(* CoDeSys 2.3 project: esx_ioxp_PPS_gazel.pro *)
(* Libraries: esx_ioxp.lib 19.12.13 13:14:40, Util.lib 18.5.10 15:14:28, Standard.lib 4.10.05 11:14:46 *)

(* PLC configuration (modules and I/O channels)
gq_Ignition AT %IX0.0 [X_SYS_IGNITION] Ignition pin (D+)
gs16_TempBoard AT %IW1 [X_SYS_TEMP_BOARD] System temperature in degree Celsius
gu32_TimeMs AT %ID1 [X_SYS_TIME_MS] System time in ms
gq_StayAlive AT %QX0.0 [X_SYS_STAY_ALIVE] Stay alive mechanism
gq_Relay AT %QX1.0 [X_SYS_RELAY_1] Safety relay
gs32_SensorSupply AT %QD1 [X_SYS_SENSOR_SUPPLY_1] External sensor supply
gs32_IO01 AT %QD2 [InOut] IO01, PIN 9 (PWM H/L, DO, CC, VIN (40V), DIN) {InOut_Type = uninitialized; InOut_FilterConfig = 0; InOut_Circuit1 = X_OUT_CIRCUIT_HIGH_SIDE; InOut_Circuit2 = X_IN_CIRCUIT_NO_PULL_UP; PWM_MaxValue = 10000}
gs32_IO02 AT %QD3 [InOut] ---- GAS meter ---- IO02, PIN 8 (PWM H/L, DO, CC, VIN (40V), DIN) {InOut_Type = X_IN_TYPE_VOLTAGE_40V; InOut_FilterConfig = 0; InOut_Circuit1 = X_IN_CIRCUIT_ACTIVE_HIGH; InOut_Circuit2 = X_IN_CIRCUIT_PULL_UP; PWM_MaxValue = 10000}
gs32_IO03 AT %QD4 [InOut] --- GAS LED BAR  ---  IO03, PIN 7 (PWM H/L, DO, CC, VIN ( {InOut_Type = X_OUT_TYPE_PWM; InOut_FilterConfig = 0; InOut_Circuit1 = X_OUT_CIRCUIT_PUSH_PULL; InOut_Circuit2 = X_IN_CIRCUIT_NO_PULL_UP; PWM_MaxValue = 10000}
gs32_IO04 AT %QD5 [InOut] IO04, PIN 6 (PWM H/L, DO, CC, VIN (40V), DIN) {InOut_Type = X_OUT_TYPE_PWM; InOut_FilterConfig = 0; InOut_Circuit1 = X_OUT_CIRCUIT_HIGH_SIDE; InOut_Circuit2 = X_IN_CIRCUIT_NO_PULL_UP; PWM_MaxValue = 10000}
gs32_IO05 AT %QD6 [InOut] IO05, PIN 13 (PWM H, DO, DIN) {InOut_Type = uninitialized; InOut_FilterConfig = 0; InOut_Circuit1 = X_OUT_CIRCUIT_HIGH_SIDE; InOut_Circuit2 = X_IN_CIRCUIT_NO_PULL_UP; PWM_MaxValue = 10000}
gs32_IO06 AT %QD7 [InOut] ---Inj1--- IO06, PIN 12 (PWM H, DO, DIN) {InOut_Type = X_OUT_TYPE_DIGITAL; InOut_FilterConfig = 0; InOut_Circuit1 = X_OUT_CIRCUIT_HIGH_SIDE; InOut_Circuit2 = X_IN_CIRCUIT_NO_PULL_UP; PWM_MaxValue = 10000}
gs32_IO07 AT %QD8 [InOut] --- Inj2 -----IO07, PIN 11 (PWM H, DO, DIN) {InOut_Type = uninitialized; InOut_FilterConfig = 0; InOut_Circuit1 = X_IN_CIRCUIT_ACTIVE_HIGH; InOut_Circuit2 = X_IN_CIRCUIT_NO_PULL_UP; PWM_MaxValue = 10000}
gs32_IO08 AT %QD9 [InOut] --- PPS1 emul --  IO08, PIN 10 (PWM H, DO, DIN) {InOut_Type = X_OUT_TYPE_PWM; InOut_FilterConfig = 0; InOut_Circuit1 = X_OUT_CIRCUIT_HIGH_SIDE; InOut_Circuit2 = X_IN_CIRCUIT_NO_PULL_UP; PWM_MaxValue = 10000}
gs32_IO09 AT %ID2 [InOut] IO09, PIN 2 (DIN, FIN, IIN) {InOut_Type = uninitialized; InOut_FilterConfig = 0; InOut_Circuit1 = X_IN_CIRCUIT_ACTIVE_HIGH; InOut_Circuit2 = X_IN_CIRCUIT_NO_PULL_UP; PWM_MaxValue = 10000}
gs32_IO10 AT %ID3 [InOut] ---RPM--- IO10, PIN 3 (DIN, FIN, IIN) {InOut_Type = X_IN_TYPE_FREQUENCY; InOut_FilterConfig = 0; InOut_Circuit1 = X_IN_CIRCUIT_ACTIVE_HIGH; InOut_Circuit2 = X_IN_CIRCUIT_NO_PULL_UP; PWM_MaxValue = 10000}
gs32_IO11 AT %ID4 [InOut] IO11, PIN 4 (DIN, FIN, IIN) {InOut_Type = uninitialized; InOut_FilterConfig = 0; InOut_Circuit1 = X_IN_CIRCUIT_ACTIVE_HIGH; InOut_Circuit2 = X_IN_CIRCUIT_NO_PULL_UP; PWM_MaxValue = 10000}
gs32_IO12 AT %ID5 [InOut] ---BLOCK ON--- IO12, PIN 5 (DIN) {InOut_Type = X_IN_TYPE_DIGITAL; InOut_FilterConfig = 0; InOut_Circuit1 = X_IN_CIRCUIT_ACTIVE_HIGH; InOut_Circuit2 = X_IN_CIRCUIT_NO_PULL_UP; PWM_MaxValue = 10000}
gs32_IO13 AT %ID6 [InOut] IO13, PIN 38 (CIN (20mA), DIN) {InOut_Type = uninitialized; InOut_FilterConfig = 0; InOut_Circuit1 = X_IN_CIRCUIT_ACTIVE_HIGH; InOut_Circuit2 = X_IN_CIRCUIT_NO_PULL_UP; PWM_MaxValue = 10000}
gs32_IO14 AT %ID7 [InOut] ---- EGR ------ IIO14, PIN 24 (CIN (20mA), DIN) {InOut_Type = X_IN_TYPE_CURRENT; InOut_FilterConfig = 0; InOut_Circuit1 = X_IN_CIRCUIT_ACTIVE_HIGH; InOut_Circuit2 = X_IN_CIRCUIT_NO_PULL_UP; PWM_MaxValue = 20000}
gs32_IO15 AT %ID8 [InOut] - Injecor temp ----IO15, PIN 39 (CIN (20mA), DIN) {InOut_Type = X_IN_TYPE_CURRENT; InOut_FilterConfig = 0; InOut_Circuit1 = X_IN_CIRCUIT_ACTIVE_HIGH; InOut_Circuit2 = X_IN_CIRCUIT_NO_PULL_UP; PWM_MaxValue = 20000}
gs32_IO16 AT %ID9 [InOut] IO16, PIN 25 (CIN (20mA), DIN) {InOut_Type = uninitialized; InOut_FilterConfig = 0; InOut_Circuit1 = X_IN_CIRCUIT_ACTIVE_HIGH; InOut_Circuit2 = X_IN_CIRCUIT_NO_PULL_UP; PWM_MaxValue = 10000}
gs32_IO17 AT %ID10 [InOut] IO17, PIN 40 (CIN (20mA), DIN) {InOut_Type = uninitialized; InOut_FilterConfig = 0; InOut_Circuit1 = X_IN_CIRCUIT_ACTIVE_HIGH; InOut_Circuit2 = X_IN_CIRCUIT_NO_PULL_UP; PWM_MaxValue = 10000}
gs32_IO18 AT %ID11 [InOut] IO18, PIN 26 (CIN (20mA), DIN) {InOut_Type = uninitialized; InOut_FilterConfig = 0; InOut_Circuit1 = X_IN_CIRCUIT_ACTIVE_HIGH; InOut_Circuit2 = X_IN_CIRCUIT_NO_PULL_UP; PWM_MaxValue = 10000}
gs32_IO19 AT %ID12 [InOut] IO19, PIN 41 (CIN (20mA), DIN) {InOut_Type = uninitialized; InOut_FilterConfig = 0; InOut_Circuit1 = X_IN_CIRCUIT_ACTIVE_HIGH; InOut_Circuit2 = X_IN_CIRCUIT_NO_PULL_UP; PWM_MaxValue = 10000}
gs32_IO20 AT %ID13 [InOut] ---Reductor_temp---  IO20, PIN 27 (CIN (20mA), DIN) {InOut_Type = X_IN_TYPE_CURRENT; InOut_FilterConfig = 0; InOut_Circuit1 = X_IN_CIRCUIT_ACTIVE_HIGH; InOut_Circuit2 = X_IN_CIRCUIT_NO_PULL_UP; PWM_MaxValue = 20000}
gs32_IO21 AT %ID14 [InOut] ---Turbo_pressure--- IO21, PIN 34 (VIN (10V), DIN) {InOut_Type = X_IN_TYPE_VOLTAGE_10V; InOut_FilterConfig = 0; InOut_Circuit1 = X_IN_CIRCUIT_ACTIVE_HIGH; InOut_Circuit2 = X_IN_CIRCUIT_NO_PULL_UP; PWM_MaxValue = 10000}
gs32_IO22 AT %ID15 [InOut] ---Reductor_press---   IO22, PIN 20 (VIN (10V), DIN) {InOut_Type = X_IN_TYPE_VOLTAGE_10V; InOut_FilterConfig = 0; InOut_Circuit1 = X_IN_CIRCUIT_ACTIVE_HIGH; InOut_Circuit2 = X_IN_CIRCUIT_NO_PULL_UP; PWM_MaxValue = 10000}
gs32_IO23 AT %ID16 [InOut] --- EGT ----IO23, PIN 35 (VIN (10V), DIN) {InOut_Type = X_IN_TYPE_VOLTAGE_10V; InOut_FilterConfig = 0; InOut_Circuit1 = X_IN_CIRCUIT_ACTIVE_HIGH; InOut_Circuit2 = X_IN_CIRCUIT_NO_PULL_UP; PWM_MaxValue = 10000}
gs32_IO24 AT %ID17 [InOut] ---PPS1--- IO24, PIN 21 (VIN (10V), DIN) {InOut_Type = uninitialized; InOut_FilterConfig = 0; InOut_Circuit1 = X_IN_CIRCUIT_ACTIVE_HIGH; InOut_Circuit2 = X_IN_CIRCUIT_NO_PULL_UP; PWM_MaxValue = 10000}
gs32_IO25 AT %ID18 [InOut] --- PPS2 ---- IO25, PIN 36 (VIN (10V), DIN) {InOut_Type = X_IN_TYPE_VOLTAGE_10V; InOut_FilterConfig = 0; InOut_Circuit1 = X_IN_CIRCUIT_ACTIVE_HIGH; InOut_Circuit2 = X_IN_CIRCUIT_NO_PULL_UP; PWM_MaxValue = 10000}
gs32_IO26 AT %ID19 [InOut] O26, PIN 22 (VIN (10V), DIN) {InOut_Type = uninitialized; InOut_FilterConfig = 0; InOut_Circuit1 = X_IN_CIRCUIT_ACTIVE_HIGH; InOut_Circuit2 = X_IN_CIRCUIT_NO_PULL_UP; PWM_MaxValue = 10000}
RS232 [X_SER_1] node 1, in %IB80 out %QB40 {X_SER_BITRATE = 19200; X_SER_STOPBITS = 1; X_SER_MODE = 8 data bits - no parity; X_SER_RX_BUFSIZE = 256; X_SER_TX_BUFSIZE = 256}
CAN1 [X_CAN_BUS_1_XC2] node 2, in %IB80 out %QB40 {X_CAN_BUS_BITRATE = 125000; X_CAN_BUS_11BIT_MASK = 16#7FF; X_CAN_BUS_29BIT_MASK = 16#1FFFFFFF}
  CAN TX Object [X_CAN_OBJ_TX_XC2] node 11771, in %IB80 out %QB40 {X_CAN_OBJ_PAUSE = 0; X_CAN_OBJ_SOFT_BUFFER = 0; X_CAN_OBJ_HARD_BUFFER = 0}
    TX AT %ID20 [X_CAN_OBJ_HANDLE] CAN object handle
  CAN RX Object [X_CAN_OBJ_RX_XC2] node 11770, in %IB84 out %QB40 {X_CAN_OBJ_ID = 16#100; X_CAN_OBJ_XTD = 11bit; X_CAN_OBJ_MASK = 16#7FF; X_CAN_OBJ_SOFT_BUFFER = 10; X_CAN_OBJ_HARD_BUFFER = 10}
    RX AT %ID21 [X_CAN_OBJ_HANDLE] CAN object handle
CAN2 [X_CAN_BUS_2_XC2] node 3, in %IB80 out %QB40 {X_CAN_BUS_BITRATE = 250000; X_CAN_BUS_11BIT_MASK = 16#7FF; X_CAN_BUS_29BIT_MASK = 16#1FFFFFFF}
*)

(* Task configuration *)
TASK Get_RPM (PRIORITY := 5, INTERVAL := T#300ms);
	Get_RPM();
END_TASK
TASK Main (PRIORITY := 20, INTERVAL := T#100ms);
	PLC_PRG();
	DFPRS_Change_Cal_Table();
	Get_Currents();
	Get_Reductor_press();
END_TASK
TASK Act_control (PRIORITY := 2, INTERVAL := T#100ms);
	Act_control();
END_TASK
TASK Get_turbo (PRIORITY := 3, INTERVAL := T#50ms);
	Get_Turbo_EGR();
END_TASK
TASK Get_key (PRIORITY := 10, INTERVAL := T#50ms);
	Get_Key();
END_TASK
TASK Emul (PRIORITY := 5, INTERVAL := T#100ms);
	Put_emul();
END_TASK
TASK Get_low_freq (PRIORITY := 5, INTERVAL := T#300ms);
	Get_EGT();
	Get_Gas_meter();
	Get_Reductor_temp();
	Get_Inj_temp();
END_TASK
TASK CAN (PRIORITY := 20, INTERVAL := T#50ms);
	Send();
	Recieve();
END_TASK

(* Global variable list: Global_Constant *)
VAR_GLOBAL CONSTANT

	TOOTH_NUM					:WORD:=58;						(* Количество зубцов на коленвале *)



	Inj_PWM_period:WORD:=250;				(* Период работы форсунок HANA=16 HZ задается в кол-ве рабочих циклов по 250 мкс*)

	(* Задание скважности PWM форсунок  ( соотношение кол-ва ЦИКЛОВ низкого сигнала к одному ВЫСОКОМУ циклу ),  *)
	(*  подбирается имперически по условию соблюдения уровня холдового тока на форсунке*)
	Inj_Low_period:WORD:=1;
	Inj_High_period:WORD:=11;
	Inj_MAX_hold_time:BYTE:=60;			(* Максимально возможная длительность холда для форсунок *)

	(* Количество срабатываний цикла обработчика прерываний, для генерирования импульса длительности открытия форсунки с пиковым током в циклах по 250 мкс*)
	Inj_peak_curent_cycle:BYTE:=16;       (* 4 мс *)

	Min_time_cnange_mode_EGT:UDINT:=60000; (* Минимальное время в мс между сменами режимов ГАЗ и ДИЗЕЛЬ для обновления статистических значений EGT *)

	PPS_tres1:INT:=20;
	PPS_tres2:INT:=100;


(*******************************************************************************************)
(*                     Настойки системы безопасности                                       *)
(*******************************************************************************************)

(*********** Пределы допустимых значений RPM ******************************)
	RPM_Min:WORD:=300;						(* Минимальный порог допкстимого RPM *)
	RPM_Max:WORD:=5500;						(* Максимальный порог допустимого RPM *)
	RPM_count:WORD:=10;						(* Максимальное количество циклов неправильного RPM, когда считаем это флуктуацией *)


	Reductor_temp_work:WORD:=4000;		(* Минимальная температура редуктора для включения блока *)
	Min_Reductor_press:WORD:=2500;		(* Минимальное давление редуктора для включения блока *)
	Min_Reductor_press_time:WORD:=40;	(*  Макстмально допустимое время минимального давления *)

	EGT_err_time:WORD:=100;					(* Через столько циклов блок опять включится что бы проверить EGT после отключения по превышению EGT *)

	Max_inj_current:DWORD:=4500000;		(* Максимальный длительный ток через газовые форсунки в микроамперах *)
	Min_inj_current:DWORD:=100;			(* Минимальный длительный ток ( обрыв ) через газовые форсунки в микроамперах *)
	Max_inj_current_time:BYTE:=5;			(* Макстмально допустимое время протекания максимального тока через форсунку в РАБОЧИХ циклах подпрограммы *)

	Inj_temp_max:DINT:=14000;				(* Максимальная температура форсунок 110 C при балластном резисторе 560 Ом* это 16000, но так как температура растет очень медленно то для подстраховки ставим 14000*)

	PPS1_min:DINT:=950;						(* Минимальный порог для PPS *)
	PPS1_max:DINT:=4300;						(* Максимальный порог для PPS *)
	PPS2_min:DINT:=450;						(* Минимальный порог для PPS *)
	PPS2_max:DINT:=2500;						(* Максимальный порог для PPS *)

(************** Конец блока безопасности ***************************************************)


END_VAR

(* Global variable list: Global_Variables *)
VAR_GLOBAL

	(* Значения считывемые с входов контролера *)

	RPM						:WORD; 				(* RPM *)
	Turbo_pressure	      :DINT;				(* Turbo pressure in mV *)
	PPS1	      			:DINT;				(* Основная педаль газа in mV *)
	OLD_PPS					:DINT;
	PPS2						:DINT;				(* Дублирующая педаль газа *)
	EGT						:DINT;				(* Температуры выхлопных газов *)
	Reductor_temp			:DINT;				(* Температура редуктора *)
	Reductor_press			:DINT;				(* Давление после редуктора *)
	Gas_meter				:DINT;				(* Давление газа *)
	Injector_temp			:DINT;				(* Температура инжекторов *)
	EGR						:DINT;				(* EGR *)

	Res_stat_pps			:BOOL;
	Min_stat_PPS			:INT;
	Max_stat_PPS			:INT;
	Avg_stat_PPS			:INT;

	(* РАЗНОЕ *)

	Inj_PWM_time			:BYTE;	 			(* Длительность холдового PWM для газового инжектора, расчитывается исходя из данных калибровки в циклах по 250 мкс*)
	Turn_start				:UDINT;				(* Системное время когда была нажата кнопка управления *)
	Count_min_reductor_press:WORD;			(* Счетчик времени для определения подлинного события падения давления в редукторе *)
	PPS1_emul				:DINT;				(* Уровень напряжения для эмулирования первой педали газа *)
	PPS2_emul				:DINT;				(* Уровень напряжения для эмулирования первой второй газа*)

	(* Структуры данных для записи в EEPROM *)

	p							:Parameters;		(* Сруктура с настройками, при старте контролера подгружаться из EEPROM*)
	a							:Always_write;		(* Структура тоже с настройками. но которая ВСЕГДА при записывается EEPROM при выключении  *)

	(* Логические переменные для включения различных режимов *)

	Flag_ECU_ON				:BOOL;				(* Контроллер включен *)
	Flag_PWM_researh		:BOOL;				(* Включения режима исследования отношения PWM к выходу операционного усилителя *)
	Flag_PPS_dyn_ON		:BOOL;
	Flag_PPS_dyn_enable	:BOOL;

	(* Логические переменные, использующиеся для обмена по CAN калибровками с питоновской прграммой *)

	Flag_CAN_send			:BOOL;				(* Запрос по CAN на посылку калибровки *)
	Flag_CAN_recieve		:BOOL;				(* Запрос по CAN на прием калибровки *)
	Flag_CAN					:BOOL;				(* Режим обмена по CAN калибровками активирован *)
	Flag_CAN_data			:BOOL;
	Flag_CAN_CRC16			:BOOL;
	Flag_CAN_Write			:BOOL;


	(*********** Флаги ошибок  *****************************)

	Err_RPM					:BOOL;				(* RPM более чем RPM_count циклов не в пределах RPM_min - RPM_max *)
	Err_EGT					:BOOL;				(* Превышен максимальный уровень EGT *)
	Err_Reductor_temp		:BOOL;				(* Недостигнута рабочая температура редуктора *)
	Err_Inj1					:BOOL;				(* Долговременно превышен максимальный ток в инжекторе 1 *)
	Err_Inj2					:BOOL;				(* Долговременно превышен максимальный ток в инжекторе 2 *)
	Err_Inj_temp			:BOOL;				(* Превышение температуры инжекторов *)
	Err_Reductor_press	:BOOL;				(* Давление в редукторе ниже нормы *)
	Err_PPS					:BOOL;				(* PPS ниже или выше допустимого значения *)

	Can_buffer				:ARRAY [1..5000] OF BYTE; 											(* Буфер для сохранения области EEPROM 400*8 *)

END_VAR

(* Data type *)
(* Эта структурв перезаписывается каждый раз при выключении *)

TYPE Always_write :
STRUCT
		Flag_byte					:BYTE;				(* 8 флагов, для хранения в EEPROM *)
		EGT_max_abs_GAS			:DINT;				(* Абсолютное максимальное достигнутое значение EGT за все время работы контроллера на ГАЗУ *)
		EGT_max_abs_DIESEL		:DINT;				(* Абсолютное максимальное достигнутое значение EGT за все время работы контроллера на ДИЗЕЛЕ *)
		EGT_max_sessions_GAS		:DINT;				(* Абсолютное максимальное значение EGT за прошлую сессию на ДИЗЕЛЕ *)
		EGT_max_sessions_DIESEL	:DINT;				(* Абсолютное максимальное значение EGT за прошлую сессию на ГАЗУ *)
END_STRUCT
END_TYPE

(* Data type *)
(* Используется для обхода ограничений по редактированию таблиц в визуализации *)

TYPE FLS :
STRUCT
	a:WORD;
END_STRUCT
END_TYPE

(* Data type *)
TYPE Parameters :

	STRUCT

		EGT_max						:WORD;						(* Максимально допустимый уровень EGT *)
		LED_BAR_PWM					:ARRAY[1..5]  OF WORD;	(* Соответствие PWM каждому диапазону датчика давления для индикатора *)
		Gas_meter_volume			:ARRAY[1..5]  OF DINT;	(* Разбивка датчика давления в баллоне на диапазоны *)
		PPS1_emul_PWM				:ARRAY[1..35] OF WORD;	(* Соответствие значения эмуляции и частотв PWM *)
		PPS_volume					:ARRAY[1..32] OF WORD;	(* Значения емуляции для каждого диапазона педали газа *)
		PPS_index					:ARRAY[1..32] OF WORD;	(* Рахзбивка педали газа на диапазоны *)
		RPM_table					:ARRAY [1..16] OF WORD;
		Turbo_table					:ARRAY [1..16] OF WORD;
		PPS_table					:ARRAY [1..16] OF WORD;
		(* Таблица для 3-х мерной калибровки *)
		Cal_table					:ARRAY [1..16,1..16,1..16] OF BYTE;
		PPS1_emul_PWM_U			:ARRAY[1..35] OF WORD;	(* Соответствие значения эмуляции и частотв PWM *)

	END_STRUCT

END_TYPE

(* POU Ввод данных/Get_RPM, ST *)
PROGRAM Get_RPM
VAR

	s16_Return   		: INT;
   Old_pulse_counter, Pulse_counter,s32_Counter    	: DINT;
   fb_InGetCounter   : FB_x_in_get_counter;

	cycle_time: DINT;
	old_time: DINT;
	i: WORD:=RPM_count;			(* Для начала работы нужно хоть одно правильное значение RPM *)
END_VAR
(* Получаем количество импульсов ( импульс=2 сигнала=открывающий и закрывающий фронт )с датчика Холла *)
fb_InGetCounter(ou16_Channel:=X_IN_10, os32_Value=>s32_Counter, os16_Status=>s16_Return);
(* Вычисляем количество импульсов за цикл работы этой прграммы *)
Pulse_counter:=s32_Counter-old_pulse_counter;
Old_pulse_counter:=s32_Counter;
(* Вычисляем время цикла в ms*)
cycle_time:=gu32_TimeMs-old_time;
old_time:=gu32_TimeMs;
(* Переводим в RPM с учетом отсутствующих зубов и времени цикла 30000=1000*60/2 *)
RPM:=DINT_TO_WORD((Pulse_counter*30000/cycle_time)/TOOTH_NUM);
(* Находится ли RPM в допустимых пределах ? *)
IF RPM<RPM_min OR RPM>RPM_max THEN
	i:=i+1;
ELSE
	i:=0;
END_IF
(* Если RPM выходит задопустимые пределы RPM_count раз подряд, тогда ошибка *)
IF i>=RPM_count THEN
	Err_RPM:=TRUE;
	i:=RPM_count;					(* Что бы избежать переполнения и ложного сброса флага *)
ELSE
	Err_RPM:=FALSE;
END_IF
END_PROGRAM

(* POU PLC_PRG, ST *)
PROGRAM PLC_PRG
VAR
	q_FirstCycle	: BOOL := TRUE;

	fb_SysClose		: FB_x_sys_close;
	fb_SsvTrigger	: FB_x_ssv_trigger;
	s16_Return,s16_Return3		: INT;

(*  Работа с входами *)
	fb_InInit    	: FB_x_in_init;
(* Работы с выходами *)
	fb_OutInit  	: FB_x_out_init;
	fb_OutSetFrequency   : FB_x_out_set_frequency;
	fb_OutSetValue   : FB_x_out_set_value;
(* Работа с таймером *)
   fb_TimClose   : FB_x_tim_close;
   fb_TimInit    : FB_x_tim_init;
   fb_TimSet     : FB_x_tim_set;
(* Работа с энергонезависимой памятью *)
	fb_EepWrite   	: FB_x_eep_write;
	fb_EepRead  	: FB_x_eep_read;

	i,k,z								:BYTE;				(* Служат для формирования байта флагов *)

	EGT_max_prev_sessions_GAS		:DINT;				(* Абсолютное максимальное значение EGT за прошлую сессию на ДИЗЕЛЕ *)
	EGT_max_prev_sessions_DIESEL	:DINT;				(* Абсолютное максимальное значение EGT за прошлую сессию на ГАЗУ *)

	Count_off: BYTE;
END_VAR
IF (q_FirstCycle = TRUE) THEN
	q_FirstCycle := FALSE;
	(* deactivate 'Safety relay' *)
	gq_Relay := FALSE;
	(* activate 'Stay alive' mechanism *)
	gq_StayAlive := TRUE;
	(* activate 'Sensor Supply' *)
	gs32_SensorSupply := X_SYS_SENSOR_SUPPLY_10V;

	Read_EEPROM();				(* Инициализируем переменные значениями из EEPROMa *)
	Init_IN();					(* Инициализируем входы *)
	Init_OUT();					(* Инициализируем выходы *)
	Init_timer();				(* Инициализируем таймер *)

	Turn_start:=gu32_TimeMs;(* Для организации паузы при включении для лога EGT *)

	(* Сохраняем значения счетчиков в целях индикации *)
	EGT_max_prev_sessions_GAS:=a.EGT_max_sessions_GAS;
	EGT_max_prev_sessions_DIESEL:=a.EGT_max_sessions_DIESEL;
	(* Для расчета максимальныйх значений именно в текущей сессии обнуляем счетчики *)
	a.EGT_max_sessions_GAS:=0;
	a.EGT_max_sessions_DIESEL:=0;

END_IF

(* trigger 'System Supervisor' *)
fb_SsvTrigger(ou16_TriggerType:=X_SSV_TRIGGER);

(* Если все условия выполняются включаем главное реле *)
IF Flag_ECU_ON AND
	Err_RPM=FALSE AND
	Err_EGT=FALSE AND
	Err_Reductor_temp=FALSE AND
	Err_Inj1=FALSE AND
	Err_inj2=FALSE AND
	Err_inj_temp=FALSE AND
	Err_PPS=FALSE AND
	Err_Reductor_press=FALSE THEN

	gq_Relay := TRUE;									(* Главное реде ВКЛ  activate 'Safety relay'*)

ELSE
	gq_Relay := FALSE;	(* Главное реде ВЫКЛ  deactivate 'Safety relay'*)
END_IF

IF (gq_Ignition = FALSE) THEN
	(* Ignition (D+) was switched off *)
	fb_TimClose(ou32_Handle:=fb_TimInit.ou32_Handle);
	(* Запакрвываем флаги в байт *)
	a.Flag_byte:=PACK(B0:=0,B1:=0,B2:=0,B3:=0,B4:=0,B5:=Flag_PPS_dyn_enable,B6:=Flag_CAN,B7:=Flag_ECU_ON);
	(* Записывем параметры газодизельного блока в энергонезависимую память *)
	fb_EepWrite(ou32_Address:=SIZEOF(p), ou32_Count:=SIZEOF(a), opu8_Data:=ADR(a), os16_Status=>s16_Return);
	(* close ESX-IOXp properly *)
	fb_SysClose();
END_IF
END_PROGRAM
ACTION Init_IN:
(**************** ИНИЦИАЛИЗАЦИЯ ВХОДОВ **************************)

(********************** Замер частоты *****************************)

(* Инициализируем вход 10, пин 3 как RPM вход *)
fb_InInit(	ou16_Channel:=X_IN_10,
        		ou16_Type:=X_IN_TYPE_FREQUENCY,
         	ou16_FilterConfig:=0,
	         ou16_InputCircuit:=X_IN_CIRCUIT_ACTIVE_HIGH,
          	ou32_CallbackParameter:=0,
	         ou16_EventCallback:=0,
          	os16_Status=>s16_Return);

(*********** Цифровой вход ********************************************)

(* Инициализируем вход 12, пин 5 как дискретный вход включения газодизельного блока  *)
fb_InInit(	ou16_Channel:=X_IN_12,
        		ou16_Type:=X_IN_TYPE_DIGITAL,
         	ou16_FilterConfig:=0,
	         ou16_InputCircuit:=X_IN_CIRCUIT_ACTIVE_HIGH,
          	ou32_CallbackParameter:=0,
	         ou16_EventCallback:=0,
          	os16_Status=>s16_Return);

(****************** Замер напряжения *****************************************)



(************************************* PPS **********************************************)
(* Инициализируем вход 24, пин 21 как вход 0..10V для основной педали газа PPS1 в mV *)
fb_InInit(	ou16_Channel:=X_IN_24,
        		ou16_Type:=X_IN_TYPE_VOLTAGE_10V,
         	ou16_FilterConfig:=0,
	         ou16_InputCircuit:=X_IN_CIRCUIT_ACTIVE_HIGH,
          	ou32_CallbackParameter:=0,
	         ou16_EventCallback:=0,
          	os16_Status=>s16_Return);

(* Инициализируем вход 25, пин 36 как вход 0..10V для PPS 2 *)
fb_InInit(	ou16_Channel:=X_IN_25,
        		ou16_Type:=X_IN_TYPE_VOLTAGE_10V,
         	ou16_FilterConfig:=0,
	         ou16_InputCircuit:=X_IN_CIRCUIT_ACTIVE_HIGH,
          	ou32_CallbackParameter:=0,
	         ou16_EventCallback:=0,
          	os16_Status=>s16_Return);
(*****************************************************************************************)

(* Инициализируем вход 21, пин 34 как вход 0..10V для Turbo pressure в mV *)
fb_InInit(	ou16_Channel:=X_IN_21,
        		ou16_Type:=X_IN_TYPE_VOLTAGE_10V,
         	ou16_FilterConfig:=0,
	         ou16_InputCircuit:=X_IN_CIRCUIT_ACTIVE_HIGH,
          	ou32_CallbackParameter:=0,
	         ou16_EventCallback:=0,
          	os16_Status=>s16_Return);


(* Инициализируем вход 22, пин 20 как вход 0..10V для Reductor press в mV *)
fb_InInit(	ou16_Channel:=X_IN_22,
        		ou16_Type:=X_IN_TYPE_VOLTAGE_10V,
         	ou16_FilterConfig:=0,
	         ou16_InputCircuit:=X_IN_CIRCUIT_ACTIVE_HIGH,
          	ou32_CallbackParameter:=0,
	         ou16_EventCallback:=0,
          	os16_Status=>s16_Return);

(* Инициализируем вход 23, пин 35 как вход 0..10V для EGT в mV *)
fb_InInit(	ou16_Channel:=X_IN_23,
        		ou16_Type:=X_IN_TYPE_VOLTAGE_10V,
         	ou16_FilterConfig:=0,
	         ou16_InputCircuit:=X_IN_CIRCUIT_ACTIVE_HIGH,
          	ou32_CallbackParameter:=0,
	         ou16_EventCallback:=0,
          	os16_Status=>s16_Return);

(* Инициализируем вход 02 , пин 08 как вход 0..40V для датчика газа в mV *)
fb_InInit(	ou16_Channel:=X_IN_02,
        		ou16_Type:=X_IN_TYPE_VOLTAGE_40V,
         	ou16_FilterConfig:=0,
	         ou16_InputCircuit:=X_IN_CIRCUIT_ACTIVE_HIGH,
          	ou32_CallbackParameter:=0,
	         ou16_EventCallback:=0,
          	os16_Status=>s16_Return);

(**************** Замер тока *******************************)

(* Инициализируем вход 20, пин 27 как токовый вход для датчика температуры редуктора  *)
fb_InInit(	ou16_Channel:=X_IN_20,
        		ou16_Type:=X_IN_TYPE_CURRENT,
         	ou16_FilterConfig:=0,
	         ou16_InputCircuit:=X_IN_CIRCUIT_ACTIVE_HIGH,
          	ou32_CallbackParameter:=0,
	         ou16_EventCallback:=0,
          	os16_Status=>s16_Return);

(* Инициализируем вход 15, пин 39 как токовый вход для датчика температуры инжекторов  *)
fb_InInit(	ou16_Channel:=X_IN_15,
        		ou16_Type:=X_IN_TYPE_CURRENT,
         	ou16_FilterConfig:=0,
	         ou16_InputCircuit:=X_IN_CIRCUIT_ACTIVE_HIGH,
          	ou32_CallbackParameter:=0,
	         ou16_EventCallback:=0,
          	os16_Status=>s16_Return);

(* Инициализируем вход 14, пин 24 как токовый вход 20 мА для EGR *)
fb_InInit(	ou16_Channel:=X_IN_24,
        		ou16_Type:=X_IN_TYPE_CURRENT,
         	ou16_FilterConfig:=0,
	         ou16_InputCircuit:=X_IN_CIRCUIT_ACTIVE_HIGH,
          	ou32_CallbackParameter:=0,
	         ou16_EventCallback:=0,
          	os16_Status=>s16_Return);
END_ACTION
ACTION Init_OUT:
(**************** ИНИЦИАЛИЗАЦИЯ ВЫХОДОВ **************************)

(* *************************  ГРУППА ВЫХОДОВ 1 **********************************************************)

(* Инициализируем выход 3, пин 7 как выход для выдачи LED *)
fb_OutInit(ou16_Channel:=X_OUT_03,
           ou16_Type:=X_OUT_TYPE_PWM +  X_OUT_CIRCUIT_HIGH_SIDE ,
           os32_MaxValue:=10000,
           ou32_CallbackParameter:=0,
           ou16_ErrorCallback:=0,
           os16_Status=>s16_Return);


(* *************************  ГРУППА ВЫХОДОВ 2 *********************************************************)


(* Инициализируем выход 6, пин 12 как выход управления Инжектором_1 *)
fb_OutInit(ou16_Channel:=X_OUT_06,
           ou16_Type:=X_OUT_TYPE_DIGITAL + X_OUT_CIRCUIT_HIGH_SIDE ,
           os32_MaxValue:=1,
           ou32_CallbackParameter:=0,
           ou16_ErrorCallback:=0,
           os16_Status=>s16_Return);

(* Инициализируем выход 7, пин 11 как выход управления Инжектором_2 *)
fb_OutInit(ou16_Channel:=X_OUT_07,
           ou16_Type:=X_OUT_TYPE_DIGITAL + X_OUT_CIRCUIT_HIGH_SIDE,
           os32_MaxValue:=1,
           ou32_CallbackParameter:=0,
           ou16_ErrorCallback:=0,
           os16_Status=>s16_Return);

(* Инициализируем выход 8, пин 10 как выход для выдачи напряжения на PPS1 *)
fb_OutInit(ou16_Channel:=X_OUT_08,
           ou16_Type:=X_OUT_TYPE_PWM +  X_OUT_CIRCUIT_HIGH_SIDE ,
           os32_MaxValue:=10000,
           ou32_CallbackParameter:=0,
           ou16_ErrorCallback:=0,
           os16_Status=>s16_Return);
END_ACTION
ACTION Init_TIMER:
(* initialize timer *)

fb_TimInit.ou16_Priority          := X_TIM_PRIO_01;
fb_TimInit.ou32_CallbackParameter := 0;
fb_TimInit.ou16_TimerCallback     := INDEXOF(TimerCallback);
fb_TimInit();
IF (fb_TimInit.os16_Status = C_NO_ERR) THEN      (* set timer *)
		fb_TimSet.ou32_Handle := fb_TimInit.ou32_Handle;
  		fb_TimSet.ou32_DelayTime := 0;
   	fb_TimSet.ou32_CycleTime := 1;
		fb_TimSet();
END_IF
END_ACTION
ACTION Read_EEPROM:
(* Читаем все параметры из энергонезависимой памяти *)
fb_EepRead(ou32_Address:=0, ou32_Count:=SIZEOF(p), opu8_Data:=ADR(p), os16_Status=>s16_Return);
fb_EepRead(ou32_Address:=SIZEOF(p), ou32_Count:=SIZEOF(a), opu8_Data:=ADR(a), os16_Status=>s16_Return);

(* Устанавливаем значение переменных, согласно битам в байте флагов *)

Flag_ECU_ON					:=EXTRACT( X:=a.Flag_byte,N:=7);				(* Биты нумеруются с 0 ! *)
Flag_CAN						:=EXTRACT( X:=a.Flag_byte,N:=6);
Flag_PPS_dyn_enable		:=EXTRACT( X:=a.Flag_byte,N:=5);
END_ACTION

(* POU TimerCallback, ST *)
PROGRAM TimerCallback
VAR
	fb_OutSetValue,fb_OutSetValue_2   : FB_x_out_set_value;
	s16_Return   	: INT;
	out: DINT;  (* Переменные в которые в прямую читаются и записываются данные с быстрых входов и выходов ПЛК 110 *)

	Peak_curent_flag: BOOL:=TRUE;	(* Флаг показывающий, что выполняется выдача пикового тока на форсунки *)
	Peak_curent_counter: WORD;		(* Счетчик циклов выдачи пикового тока на форсунки *)

	Hold_curent_low_counter:WORD;		(* Счетчик циклов выдачи низкого уровня в цикле выдачи холдового тока на форсунки *)
	Hold_curent_High_counter: WORD;

	Hold_curent_counter:WORD;			(* Счетчик циклов выдачи холдового тока на форсунки *)
	Hold_curent_flag: BOOL;			(* Флаг показывающий, что выполняется выдача тока удержаня на газовые форсунки *)

	Inj_Big_cycle: WORD; 				(* Счетчик выполненных циклов в  большом цикле работы форсунок HANA=10 Hz *)
	Inj_hold_High_flag: BOOL;

	Act_PWM_High_flag: BOOL;
	Act_PWM_High_counter: WORD;
	Act_PWM_Low_counter: WORD;
END_VAR
(* Форсунки фключаются только когда газ и блок включены и имеется холд ток и не включен спецрежи выключения блока *)
IF Flag_ECU_ON AND Inj_PWM_time > 0 THEN
				IF Inj_Big_cycle<Inj_PWM_period THEN			(* Большой цикл работы форсунок, длительность которого  Inj_PWM_period установлена производителем. куда входит пиковый ток, холд ток и пауза *)
						Inj_Big_cycle:=Inj_Big_cycle+1;
						(* Выдача пикового тока *)
						IF Peak_curent_flag=TRUE THEN
								IF Peak_curent_counter< Inj_peak_curent_cycle THEN (*  Длительность выдачи пикового тока на форсунки Inj_peak_curent_cycle устанавливается производителем задается в разделе констант*)
										Peak_curent_counter:=Peak_curent_counter+1;
										out:=1;
								ELSE
										Peak_curent_counter:=0;
										out:=0;
										Peak_curent_flag:=FALSE;
								END_IF
						ELSIF Hold_curent_flag=TRUE THEN
								(********** Выдача тока удержания *)
								IF Hold_curent_counter<Inj_PWM_time THEN                (* Длительность выдачи тока удержания Inj_PWM_time, выраженная в кол-ве циклов обработчика прерывания вычисляется из данных  калибровочной таблицы *)
										Hold_curent_counter:=Hold_curent_counter+1;
										IF Inj_hold_High_flag=TRUE THEN									(*  Идет генерация импульса высокого уровня *)
												IF Hold_curent_High_counter < Inj_High_period THEN
														Hold_curent_High_counter:=Hold_curent_High_counter+1;
														out:=1;
												ELSE
														out:=0;
														Inj_hold_High_flag:=FALSE;
														Hold_curent_Low_counter:=1;
												END_IF
										ELSE																	(* Идет генерация пауз между имплусами высокого уровня *)
												IF Hold_curent_Low_counter < Inj_Low_period THEN
														Hold_curent_Low_counter:=Hold_curent_Low_counter+1;
														out:=0;
												ELSE
														Inj_hold_High_flag:=TRUE;
														Hold_curent_High_counter:=1;
														out:=1;
												END_IF
										END_IF
								ELSE
										Hold_curent_counter:=0;
										Hold_curent_flag:=FALSE;
										out:=0;
								END_IF
						END_IF
				ELSE
						Inj_Big_cycle:=0;
						Peak_curent_flag:=TRUE;
						Hold_curent_flag:=TRUE;
				END_IF
		(* Прямое управление выходами для инжекторов *)
		fb_OutSetValue(ou16_Channel:=X_OUT_06, os32_Value:=out, os16_Status=>s16_Return);
		fb_OutSetValue(ou16_Channel:=X_OUT_07, os32_Value:=out, os16_Status=>s16_Return);
ELSE
		(* На всякий случай явно выключим инжекторы, если не выполняются условия их включения *)
		fb_OutSetValue(ou16_Channel:=X_OUT_06, os32_Value:=0, os16_Status=>s16_Return);
		fb_OutSetValue(ou16_Channel:=X_OUT_07, os32_Value:=0, os16_Status=>s16_Return);
END_IF
END_PROGRAM

(* POU DFPRS_Change_Cal_Table, ST *)
PROGRAM DFPRS_Change_Cal_Table
VAR
	(* Флаги для инициализации различных действий из визуализации *)
	(* для всей таблицы *)
	Write_cal, Read_cal	:BOOL; (* Считать или записать данные в EEPROM *)
	Write_cal2,Red_cal2	:BOOL; (* Считать или записать данные из таблицы в окно редактора *)
	HALF_set_ALL,Set_ALL	:BOOL;
	ALL_plus, ALL_minus	:BOOL;

	(* для RPM *)
	RPM_Flag_plus_1,RPM_Flag_plus_2,RPM_Flag_plus_3,RPM_Flag_plus_4,RPM_Flag_plus_5,RPM_Flag_plus_6,RPM_Flag_plus_7,RPM_Flag_plus_8:BOOL;
	RPM_Flag_plus_9,RPM_Flag_plus_10,RPM_Flag_plus_11,RPM_Flag_plus_12,RPM_Flag_plus_13,RPM_Flag_plus_14,RPM_Flag_plus_15,RPM_Flag_plus_16:BOOL;

	RPM_Flag_minus_1,RPM_Flag_minus_2,RPM_Flag_minus_3,RPM_Flag_minus_4,RPM_Flag_minus_5,RPM_Flag_minus_6,RPM_Flag_minus_7,RPM_Flag_minus_8:BOOL;
	RPM_Flag_minus_9,RPM_Flag_minus_10,RPM_Flag_minus_11,RPM_Flag_minus_12,RPM_Flag_minus_13,RPM_Flag_minus_14,RPM_Flag_minus_15,RPM_Flag_minus_16:BOOL;

	RPM_Flag_CP_1,RPM_Flag_CP_2,RPM_Flag_CP_3,RPM_Flag_CP_4,RPM_Flag_CP_5,RPM_Flag_CP_6,RPM_Flag_CP_7,RPM_Flag_CP_8:BOOL;
	RPM_Flag_CP_9,RPM_Flag_CP_10,RPM_Flag_CP_11,RPM_Flag_CP_12,RPM_Flag_CP_13,RPM_Flag_CP_14,RPM_Flag_CP_15,RPM_Flag_CP_16:BOOL;

	(* для Turbo *)
	Turbo_Flag_plus_1,Turbo_Flag_plus_2,Turbo_Flag_plus_3,Turbo_Flag_plus_4,Turbo_Flag_plus_5,Turbo_Flag_plus_6,Turbo_Flag_plus_7,Turbo_Flag_plus_8:BOOL;
	Turbo_Flag_plus_9,Turbo_Flag_plus_10,Turbo_Flag_plus_11,Turbo_Flag_plus_12,Turbo_Flag_plus_13,Turbo_Flag_plus_14,Turbo_Flag_plus_15,Turbo_Flag_plus_16:BOOL;

	Turbo_Flag_minus_1,Turbo_Flag_minus_2,Turbo_Flag_minus_3,Turbo_Flag_minus_4,Turbo_Flag_minus_5,Turbo_Flag_minus_6,Turbo_Flag_minus_7,Turbo_Flag_minus_8:BOOL;
	Turbo_Flag_minus_9,Turbo_Flag_minus_10,Turbo_Flag_minus_11,Turbo_Flag_minus_12,Turbo_Flag_minus_13,Turbo_Flag_minus_14,Turbo_Flag_minus_15,Turbo_Flag_minus_16:BOOL;

	Turbo_Flag_CP_1,Turbo_Flag_CP_2,Turbo_Flag_CP_3,Turbo_Flag_CP_4,Turbo_Flag_CP_5,Turbo_Flag_CP_6,Turbo_Flag_CP_7,Turbo_Flag_CP_8:BOOL;
	Turbo_Flag_CP_9,Turbo_Flag_CP_10,Turbo_Flag_CP_11,Turbo_Flag_CP_12,Turbo_Flag_CP_13,Turbo_Flag_CP_14,Turbo_Flag_CP_15,Turbo_Flag_CP_16:BOOL;

	(* Выбор типа калибровки и диапазона PPS *)
	PPS_number:BYTE;				(* Может принимать значение от 1 до 8 по числу диапазонов PPS *)

	(* Буферный массив с которым идет работа, а потом он копируется в калибровку *)
	Buffer: ARRAY [1..16,1..16] OF FLS;

	i,j,k:BYTE;
	z:WORD;

	Change_volume:WORD:=10;


	s16_Return    	: INT;
	fb_EepWrite   	: FB_x_eep_write;
	fb_EepRead  	: FB_x_eep_read;

END_VAR
(*********************** Работа с главной калибровочной таблицей ********************************************)

(* Сохраняем или читаем калибровку в/из EEPROM *)
EEPROM_read_write();
(* Считать требуемые данные из калибровочной таблицы в окно редактора *)
Buffer_read_write();
(* Обработка данных в окне буфера: увеличить все, уменьшить все, залить значение и т.д *)
Edit_function();

(***************************************** RPM ********************************************************)

(* Добавляем фиксированное значение к текущему значению в строке RPM *)
RPM_plus();
(* Вычитаем фиксированное значение к текущему значению в строке RPM *)
RPM_minus();
(* Копируем предидущую строку RPM в текущую *)
RPM_copy();

(********************************************TURBO*****************************************************)

(* Добавляем фиксированное значение к текущему значению в столбце Turbo *)
Turbo_plus();
(* Вычитаем фиксированное значение к текущему значению в столбце TURBO *)
Turbo_minus();
(* Копируем предидущий столбец Tubor в текущий *)
Turbo_copy();
END_PROGRAM
ACTION Buffer_read_write:
(* Считать требуемые данные из калибровочной таблицы в окно редактора *)
IF Red_cal2 THEN

				FOR i:=1 TO 16 DO
					FOR j:=1 TO 16 DO
						Buffer[i,j].a:=p.Cal_table[i,j,PPS_number];
					END_FOR
				END_FOR

	Red_cal2:=FALSE;
END_IF

(* Записать текущие данные из окна редактора в калибровочную таблицу *)
IF Write_cal2 THEN

				FOR i:=1 TO 16 DO
					FOR j:=1 TO 16 DO
						p.Cal_table[i,j,PPS_number]:=WORD_TO_BYTE(Buffer[i,j].a);
					END_FOR
				END_FOR

	Write_cal2:=FALSE;
END_IF
END_ACTION
ACTION Edit_function:
(* Устанавливаем в определенное значение все значения в окне редактора *)
IF Set_ALL THEN
				FOR i:=1 TO 16 DO
						FOR j:=1 TO 16 DO
							Buffer[i,j].a:=Change_volume;
						END_FOR
				END_FOR
	Set_ALL:=FALSE;
END_IF

(* Устанавливаем в определенное значение нижнюю диагональ  в окне редактора *)
IF HALF_set_ALL THEN
				k:=17;
				i:=17;
				FOR j:=1 TO 16 DO
					k:=k-1;
					i:=17;
						WHILE i<>k  DO
							i:=i-1;
							Buffer[i,j].a:=Change_volume;
						END_WHILE
				END_FOR
	HALF_set_ALL:=FALSE;
END_IF

(* Увеличиваем все значения  в окне редактора *)
IF ALL_plus THEN
				FOR i:=1 TO 16 DO
						FOR j:=1 TO 16 DO
							Buffer[i,j].a:=Buffer[i,j].a+Change_volume;
						END_FOR
				END_FOR
	ALL_plus:=FALSE;
END_IF

(* Уменьшаем все значения  в окне редактора *)

IF ALL_minus THEN
				FOR i:=1 TO 16 DO
						FOR j:=1 TO 16 DO
							Buffer[i,j].a:=Buffer[i,j].a-Change_volume;
						END_FOR
				END_FOR
	ALL_minus:=FALSE;
END_IF
END_ACTION
ACTION EEPROM_read_write:
(* Сохраняем калибровку в файле *)
IF Write_Cal THEN
	fb_EepWrite(ou32_Address:=0, ou32_Count:=SIZEOF(p), opu8_Data:=ADR(p), os16_Status=>s16_Return);
	Write_cal:=FALSE;
END_IF

(* Читаем калибровку из файла *)
IF Read_Cal THEN
	fb_EepRead(ou32_Address:=0, ou32_Count:=SIZEOF(p), opu8_Data:=ADR(p), os16_Status=>s16_Return);
	Read_cal:=FALSE;
END_IF
END_ACTION
ACTION RPM_copy:
(* Копируем предидущую строку RPM в текущую *)

IF RPM_Flag_CP_2 THEN
	FOR i:=1 TO 16 DO
		Buffer[i,2].a:=Buffer[i,1].a;
	END_FOR
	RPM_Flag_CP_2:=FALSE;
END_IF
IF RPM_Flag_CP_3 THEN
	FOR i:=1 TO 16 DO
		Buffer[i,3].a:=Buffer[i,2].a;
	END_FOR
	RPM_Flag_CP_3:=FALSE;
END_IF
IF RPM_Flag_CP_4 THEN
	FOR i:=1 TO 16 DO
		Buffer[i,4].a:=Buffer[i,3].a;
	END_FOR
	RPM_Flag_CP_4:=FALSE;
END_IF
IF RPM_Flag_CP_5 THEN
	FOR i:=1 TO 16 DO
		Buffer[i,5].a:=Buffer[i,4].a;
	END_FOR
	RPM_Flag_CP_5:=FALSE;
END_IF
IF RPM_Flag_CP_6 THEN
	FOR i:=1 TO 16 DO
		Buffer[i,6].a:=Buffer[i,5].a;
	END_FOR
	RPM_Flag_CP_6:=FALSE;
END_IF
IF RPM_Flag_CP_7 THEN
	FOR i:=1 TO 16 DO
		Buffer[i,7].a:=Buffer[i,6].a;
	END_FOR
	RPM_Flag_CP_7:=FALSE;
END_IF
IF RPM_Flag_CP_8 THEN
	FOR i:=1 TO 16 DO
		Buffer[i,8].a:=Buffer[i,7].a;
	END_FOR
	RPM_Flag_CP_8:=FALSE;
END_IF

IF RPM_Flag_CP_9 THEN
	FOR i:=1 TO 16 DO
		Buffer[i,9].a:=Buffer[i,8].a;
	END_FOR
	RPM_Flag_CP_9:=FALSE;
END_IF
IF RPM_Flag_CP_10 THEN
	FOR i:=1 TO 16 DO
		Buffer[i,10].a:=Buffer[i,9].a;
	END_FOR
	RPM_Flag_CP_10:=FALSE;
END_IF
IF RPM_Flag_CP_11 THEN
	FOR i:=1 TO 16 DO
		Buffer[i,11].a:=Buffer[i,10].a;
	END_FOR
	RPM_Flag_CP_11:=FALSE;
END_IF
IF RPM_Flag_CP_12 THEN
	FOR i:=1 TO 16 DO
		Buffer[i,12].a:=Buffer[i,11].a;
	END_FOR
	RPM_Flag_CP_12:=FALSE;
END_IF
IF RPM_Flag_CP_13 THEN
	FOR i:=1 TO 16 DO
		Buffer[i,13].a:=Buffer[i,12].a;
	END_FOR
	RPM_Flag_CP_13:=FALSE;
END_IF
IF RPM_Flag_CP_14 THEN
	FOR i:=1 TO 16 DO
		Buffer[i,14].a:=Buffer[i,13].a;
	END_FOR
	RPM_Flag_CP_14:=FALSE;
END_IF
IF RPM_Flag_CP_15 THEN
	FOR i:=1 TO 16 DO
		Buffer[i,15].a:=Buffer[i,14].a;
	END_FOR
	RPM_Flag_CP_15:=FALSE;
END_IF

IF RPM_Flag_CP_16 THEN
	FOR i:=1 TO 16 DO
		Buffer[i,16].a:=Buffer[i,15].a;
	END_FOR
	RPM_Flag_CP_16:=FALSE;
END_IF
END_ACTION
ACTION RPM_minus:
(* Вычитаем фиксированное значение к текущему значению в строке RPM *)

IF RPM_Flag_minus_1 THEN
	FOR i:=1 TO 16 DO
		Buffer[i,1].a:=Buffer[i,1].a-Change_volume;
	END_FOR
	RPM_Flag_minus_1:=FALSE;
END_IF
IF RPM_Flag_minus_2 THEN
	FOR i:=1 TO 16 DO
		Buffer[i,2].a:=Buffer[i,2].a-Change_volume;
	END_FOR
	RPM_Flag_minus_2:=FALSE;
END_IF
IF RPM_Flag_minus_3 THEN
	FOR i:=1 TO 16 DO
		Buffer[i,3].a:=Buffer[i,3].a-Change_volume;
	END_FOR
	RPM_Flag_minus_3:=FALSE;
END_IF
IF RPM_Flag_minus_4 THEN
	FOR i:=1 TO 16 DO
		Buffer[i,4].a:=Buffer[i,4].a-Change_volume;
	END_FOR
	RPM_Flag_minus_4:=FALSE;
END_IF
IF RPM_Flag_minus_5 THEN
	FOR i:=1 TO 16 DO
		Buffer[i,5].a:=Buffer[i,5].a-Change_volume;
	END_FOR
	RPM_Flag_minus_5:=FALSE;
END_IF
IF RPM_Flag_minus_6 THEN
	FOR i:=1 TO 16 DO
		Buffer[i,6].a:=Buffer[i,6].a-Change_volume;
	END_FOR
	RPM_Flag_minus_6:=FALSE;
END_IF
IF RPM_Flag_minus_7 THEN
	FOR i:=1 TO 16 DO
		Buffer[i,7].a:=Buffer[i,7].a-Change_volume;
	END_FOR
	RPM_Flag_minus_7:=FALSE;
END_IF
IF RPM_Flag_minus_8 THEN
	FOR i:=1 TO 16 DO
		Buffer[i,8].a:=Buffer[i,8].a-Change_volume;
	END_FOR
	RPM_Flag_minus_8:=FALSE;
END_IF

IF RPM_Flag_minus_9 THEN
	FOR i:=1 TO 16 DO
		Buffer[i,9].a:=Buffer[i,9].a-Change_volume;
	END_FOR
	RPM_Flag_minus_9:=FALSE;
END_IF
IF RPM_Flag_minus_10 THEN
	FOR i:=1 TO 16 DO
		Buffer[i,10].a:=Buffer[i,10].a-Change_volume;
	END_FOR
	RPM_Flag_minus_10:=FALSE;
END_IF
IF RPM_Flag_minus_11 THEN
	FOR i:=1 TO 16 DO
		Buffer[i,11].a:=Buffer[i,11].a-Change_volume;
	END_FOR
	RPM_Flag_minus_11:=FALSE;
END_IF
IF RPM_Flag_minus_12 THEN
	FOR i:=1 TO 16 DO
		Buffer[i,12].a:=Buffer[i,12].a-Change_volume;
	END_FOR
	RPM_Flag_minus_12:=FALSE;
END_IF
IF RPM_Flag_minus_13 THEN
	FOR i:=1 TO 16 DO
		Buffer[i,13].a:=Buffer[i,13].a-Change_volume;
	END_FOR
	RPM_Flag_minus_13:=FALSE;
END_IF
IF RPM_Flag_minus_14 THEN
	FOR i:=1 TO 16 DO
		Buffer[i,14].a:=Buffer[i,14].a-Change_volume;
	END_FOR
	RPM_Flag_minus_14:=FALSE;
END_IF
IF RPM_Flag_minus_15 THEN
	FOR i:=1 TO 16 DO
		Buffer[i,15].a:=Buffer[i,15].a-Change_volume;
	END_FOR
	RPM_Flag_minus_15:=FALSE;
END_IF
IF RPM_Flag_minus_16 THEN
	FOR i:=1 TO 16 DO
		Buffer[i,16].a:=Buffer[i,16].a-Change_volume;
	END_FOR
	RPM_Flag_minus_16:=FALSE;
END_IF
END_ACTION
ACTION RPM_plus:
(* Добавляем фиксированное значение к текущему значению в строке RPM *)

IF RPM_Flag_plus_1 THEN
	FOR i:=1 TO 16 DO
		Buffer[i,1].a:=Buffer[i,1].a+Change_volume;
	END_FOR
	RPM_Flag_plus_1:=FALSE;
END_IF
IF RPM_Flag_plus_2 THEN
	FOR i:=1 TO 16 DO
		Buffer[i,2].a:=Buffer[i,2].a+Change_volume;
	END_FOR
	RPM_Flag_plus_2:=FALSE;
END_IF
IF RPM_Flag_plus_3 THEN
	FOR i:=1 TO 16 DO
		Buffer[i,3].a:=Buffer[i,3].a+Change_volume;
	END_FOR
	RPM_Flag_plus_3:=FALSE;
END_IF
IF RPM_Flag_plus_4 THEN
	FOR i:=1 TO 16 DO
		Buffer[i,4].a:=Buffer[i,4].a+Change_volume;
	END_FOR
	RPM_Flag_plus_4:=FALSE;
END_IF
IF RPM_Flag_plus_5 THEN
	FOR i:=1 TO 16 DO
		Buffer[i,5].a:=Buffer[i,5].a+Change_volume;
	END_FOR
	RPM_Flag_plus_5:=FALSE;
END_IF
IF RPM_Flag_plus_6 THEN
	FOR i:=1 TO 16 DO
		Buffer[i,6].a:=Buffer[i,6].a+Change_volume;
	END_FOR
	RPM_Flag_plus_6:=FALSE;
END_IF
IF RPM_Flag_plus_7 THEN
	FOR i:=1 TO 16 DO
		Buffer[i,7].a:=Buffer[i,7].a+Change_volume;
	END_FOR
	RPM_Flag_plus_7:=FALSE;
END_IF
IF RPM_Flag_plus_8 THEN
	FOR i:=1 TO 16 DO
		Buffer[i,8].a:=Buffer[i,8].a+Change_volume;
	END_FOR
	RPM_Flag_plus_8:=FALSE;
END_IF


IF RPM_Flag_plus_9 THEN
	FOR i:=1 TO 16 DO
		Buffer[i,9].a:=Buffer[i,9].a+Change_volume;
	END_FOR
	RPM_Flag_plus_9:=FALSE;
END_IF
IF RPM_Flag_plus_10 THEN
	FOR i:=1 TO 16 DO
		Buffer[i,10].a:=Buffer[i,10].a+Change_volume;
	END_FOR
	RPM_Flag_plus_10:=FALSE;
END_IF
IF RPM_Flag_plus_11 THEN
	FOR i:=1 TO 16 DO
		Buffer[i,11].a:=Buffer[i,11].a+Change_volume;
	END_FOR
	RPM_Flag_plus_11:=FALSE;
END_IF
IF RPM_Flag_plus_12 THEN
	FOR i:=1 TO 16 DO
		Buffer[i,12].a:=Buffer[i,12].a+Change_volume;
	END_FOR
	RPM_Flag_plus_12:=FALSE;
END_IF
IF RPM_Flag_plus_13 THEN
	FOR i:=1 TO 16 DO
		Buffer[i,13].a:=Buffer[i,13].a+Change_volume;
	END_FOR
	RPM_Flag_plus_13:=FALSE;
END_IF
IF RPM_Flag_plus_14 THEN
	FOR i:=1 TO 16 DO
		Buffer[i,14].a:=Buffer[i,14].a+Change_volume;
	END_FOR
	RPM_Flag_plus_14:=FALSE;
END_IF
IF RPM_Flag_plus_15 THEN
	FOR i:=1 TO 16 DO
		Buffer[i,15].a:=Buffer[i,15].a+Change_volume;
	END_FOR
	RPM_Flag_plus_15:=FALSE;
END_IF
IF RPM_Flag_plus_16 THEN
	FOR i:=1 TO 16 DO
		Buffer[i,16].a:=Buffer[i,16].a+Change_volume;
	END_FOR
	RPM_Flag_plus_16:=FALSE;
END_IF
END_ACTION
ACTION Turbo_copy:
(* Копируем предидущий столбец Tubor в текущий *)

IF Turbo_Flag_CP_2 THEN
	FOR i:=1 TO 16 DO
		Buffer[2,i].a:=Buffer[1,i].a;
	END_FOR
	Turbo_Flag_CP_2:=FALSE;
END_IF
IF Turbo_Flag_CP_3 THEN
	FOR i:=1 TO 16 DO
		Buffer[3,i].a:=Buffer[2,i].a;
	END_FOR
	Turbo_Flag_CP_3:=FALSE;
END_IF
IF Turbo_Flag_CP_4 THEN
	FOR i:=1 TO 16 DO
		Buffer[4,i].a:=Buffer[3,i].a;
	END_FOR
	Turbo_Flag_CP_4:=FALSE;
END_IF
IF Turbo_Flag_CP_5 THEN
	FOR i:=1 TO 16 DO
		Buffer[5,i].a:=Buffer[4,i].a;
	END_FOR
	Turbo_Flag_CP_5:=FALSE;
END_IF
IF Turbo_Flag_CP_6 THEN
	FOR i:=1 TO 16 DO
		Buffer[6,i].a:=Buffer[5,i].a;
	END_FOR
	Turbo_Flag_CP_6:=FALSE;
END_IF
IF Turbo_Flag_CP_7 THEN
	FOR i:=1 TO 16 DO
		Buffer[7,i].a:=Buffer[6,i].a;
	END_FOR
	Turbo_Flag_CP_7:=FALSE;
END_IF
IF Turbo_Flag_CP_8 THEN
	FOR i:=1 TO 8 DO
		Buffer[8,i].a:=Buffer[7,i].a;
	END_FOR
	Turbo_Flag_CP_8:=FALSE;
END_IF

IF Turbo_Flag_CP_9 THEN
	FOR i:=1 TO 16 DO
		Buffer[9,i].a:=Buffer[8,i].a;
	END_FOR
	Turbo_Flag_CP_9:=FALSE;
END_IF
IF Turbo_Flag_CP_10 THEN
	FOR i:=1 TO 16 DO
		Buffer[10,i].a:=Buffer[9,i].a;
	END_FOR
	Turbo_Flag_CP_10:=FALSE;
END_IF
IF Turbo_Flag_CP_11 THEN
	FOR i:=1 TO 16 DO
		Buffer[11,i].a:=Buffer[10,i].a;
	END_FOR
	Turbo_Flag_CP_11:=FALSE;
END_IF
IF Turbo_Flag_CP_12 THEN
	FOR i:=1 TO 16 DO
		Buffer[12,i].a:=Buffer[11,i].a;
	END_FOR
	Turbo_Flag_CP_12:=FALSE;
END_IF
IF Turbo_Flag_CP_13 THEN
	FOR i:=1 TO 16 DO
		Buffer[13,i].a:=Buffer[12,i].a;
	END_FOR
	Turbo_Flag_CP_13:=FALSE;
END_IF
IF Turbo_Flag_CP_14 THEN
	FOR i:=1 TO 16 DO
		Buffer[14,i].a:=Buffer[13,i].a;
	END_FOR
	Turbo_Flag_CP_14:=FALSE;
END_IF
IF Turbo_Flag_CP_15 THEN
	FOR i:=1 TO 8 DO
		Buffer[15,i].a:=Buffer[14,i].a;
	END_FOR
	Turbo_Flag_CP_15:=FALSE;
END_IF
IF Turbo_Flag_CP_16 THEN
	FOR i:=1 TO 8 DO
		Buffer[16,i].a:=Buffer[15,i].a;
	END_FOR
	Turbo_Flag_CP_16:=FALSE;
END_IF
END_ACTION
ACTION Turbo_minus:
(* Вычитаем фиксированное значение к текущему значению в столбце TURBO *)

IF Turbo_Flag_minus_1 THEN
	FOR i:=1 TO 16 DO
		Buffer[1,i].a:=Buffer[1,i].a-Change_volume;
	END_FOR
	Turbo_Flag_minus_1:=FALSE;
END_IF
IF Turbo_Flag_minus_2 THEN
	FOR i:=1 TO 16 DO
		Buffer[2,i].a:=Buffer[2,i].a-Change_volume;
	END_FOR
	Turbo_Flag_minus_2:=FALSE;
END_IF
IF Turbo_Flag_minus_3 THEN
	FOR i:=1 TO 16 DO
		Buffer[3,i].a:=Buffer[3,i].a-Change_volume;
	END_FOR
	Turbo_Flag_minus_3:=FALSE;
END_IF
IF Turbo_Flag_minus_4 THEN
	FOR i:=1 TO 16 DO
		Buffer[4,i].a:=Buffer[4,i].a-Change_volume;
	END_FOR
	Turbo_Flag_minus_4:=FALSE;
END_IF
IF Turbo_Flag_minus_5 THEN
	FOR i:=1 TO 16 DO
		Buffer[5,i].a:=Buffer[5,i].a-Change_volume;
	END_FOR
	Turbo_Flag_minus_5:=FALSE;
END_IF
IF Turbo_Flag_minus_6 THEN
	FOR i:=1 TO 16 DO
		Buffer[6,i].a:=Buffer[6,i].a-Change_volume;
	END_FOR
	Turbo_Flag_minus_6:=FALSE;
END_IF
IF Turbo_Flag_minus_7 THEN
	FOR i:=1 TO 16 DO
		Buffer[7,i].a:=Buffer[7,i].a-Change_volume;
	END_FOR
	Turbo_Flag_minus_7:=FALSE;
END_IF
IF Turbo_Flag_minus_8 THEN
	FOR i:=1 TO 16 DO
		Buffer[8,i].a:=Buffer[8,i].a-Change_volume;
	END_FOR
	Turbo_Flag_minus_8:=FALSE;
END_IF

IF Turbo_Flag_minus_9 THEN
	FOR i:=1 TO 16 DO
		Buffer[9,i].a:=Buffer[9,i].a-Change_volume;
	END_FOR
	Turbo_Flag_minus_9:=FALSE;
END_IF
IF Turbo_Flag_minus_10 THEN
	FOR i:=1 TO 16 DO
		Buffer[10,i].a:=Buffer[10,i].a-Change_volume;
	END_FOR
	Turbo_Flag_minus_10:=FALSE;
END_IF
IF Turbo_Flag_minus_11 THEN
	FOR i:=1 TO 16 DO
		Buffer[11,i].a:=Buffer[11,i].a-Change_volume;
	END_FOR
	Turbo_Flag_minus_11:=FALSE;
END_IF
IF Turbo_Flag_minus_12 THEN
	FOR i:=1 TO 16 DO
		Buffer[12,i].a:=Buffer[12,i].a-Change_volume;
	END_FOR
	Turbo_Flag_minus_12:=FALSE;
END_IF
IF Turbo_Flag_minus_13 THEN
	FOR i:=1 TO 16 DO
		Buffer[13,i].a:=Buffer[13,i].a-Change_volume;
	END_FOR
	Turbo_Flag_minus_13:=FALSE;
END_IF
IF Turbo_Flag_minus_14 THEN
	FOR i:=1 TO 16 DO
		Buffer[14,i].a:=Buffer[14,i].a-Change_volume;
	END_FOR
	Turbo_Flag_minus_14:=FALSE;
END_IF
IF Turbo_Flag_minus_15 THEN
	FOR i:=1 TO 16 DO
		Buffer[15,i].a:=Buffer[15,i].a-Change_volume;
	END_FOR
	Turbo_Flag_minus_15:=FALSE;
END_IF
IF Turbo_Flag_minus_16 THEN
	FOR i:=1 TO 16 DO
		Buffer[16,i].a:=Buffer[16,i].a-Change_volume;
	END_FOR
	Turbo_Flag_minus_16:=FALSE;
END_IF
END_ACTION
ACTION Turbo_plus:
(* Добавляем фиксированное значение к текущему значению в столбце Turbo *)

IF Turbo_Flag_plus_1 THEN
	FOR i:=1 TO 16 DO
		Buffer[1,i].a:=Buffer[1,i].a+Change_volume;
	END_FOR
	Turbo_Flag_plus_1:=FALSE;
END_IF
IF Turbo_Flag_plus_2 THEN
	FOR i:=1 TO 16 DO
		Buffer[2,i].a:=Buffer[2,i].a+Change_volume;
	END_FOR
	Turbo_Flag_plus_2:=FALSE;
END_IF
IF Turbo_Flag_plus_3 THEN
	FOR i:=1 TO 16 DO
		Buffer[3,i].a:=Buffer[3,i].a+Change_volume;
	END_FOR
	Turbo_Flag_plus_3:=FALSE;
END_IF
IF Turbo_Flag_plus_4 THEN
	FOR i:=1 TO 16 DO
		Buffer[4,i].a:=Buffer[4,i].a+Change_volume;
	END_FOR
	Turbo_Flag_plus_4:=FALSE;
END_IF
IF Turbo_Flag_plus_5 THEN
	FOR i:=1 TO 16 DO
		Buffer[5,i].a:=Buffer[5,i].a+Change_volume;
	END_FOR
	Turbo_Flag_plus_5:=FALSE;
END_IF
IF Turbo_Flag_plus_6 THEN
	FOR i:=1 TO 16 DO
		Buffer[6,i].a:=Buffer[6,i].a+Change_volume;
	END_FOR
	Turbo_Flag_plus_6:=FALSE;
END_IF
IF Turbo_Flag_plus_7 THEN
	FOR i:=1 TO 16 DO
		Buffer[7,i].a:=Buffer[7,i].a+Change_volume;
	END_FOR
	Turbo_Flag_plus_7:=FALSE;
END_IF
IF Turbo_Flag_plus_8 THEN
	FOR i:=1 TO 16 DO
		Buffer[8,i].a:=Buffer[8,i].a+Change_volume;
	END_FOR
	Turbo_Flag_plus_8:=FALSE;
END_IF

IF Turbo_Flag_plus_9 THEN
	FOR i:=1 TO 16 DO
		Buffer[9,i].a:=Buffer[9,i].a+Change_volume;
	END_FOR
	Turbo_Flag_plus_9:=FALSE;
END_IF
IF Turbo_Flag_plus_10 THEN
	FOR i:=1 TO 16 DO
		Buffer[10,i].a:=Buffer[10,i].a+Change_volume;
	END_FOR
	Turbo_Flag_plus_10:=FALSE;
END_IF
IF Turbo_Flag_plus_11 THEN
	FOR i:=1 TO 16 DO
		Buffer[11,i].a:=Buffer[11,i].a+Change_volume;
	END_FOR
	Turbo_Flag_plus_11:=FALSE;
END_IF
IF Turbo_Flag_plus_12 THEN
	FOR i:=1 TO 16 DO
		Buffer[12,i].a:=Buffer[12,i].a+Change_volume;
	END_FOR
	Turbo_Flag_plus_12:=FALSE;
END_IF
IF Turbo_Flag_plus_13 THEN
	FOR i:=1 TO 16 DO
		Buffer[13,i].a:=Buffer[13,i].a+Change_volume;
	END_FOR
	Turbo_Flag_plus_13:=FALSE;
END_IF
IF Turbo_Flag_plus_14 THEN
	FOR i:=1 TO 16 DO
		Buffer[14,i].a:=Buffer[14,i].a+Change_volume;
	END_FOR
	Turbo_Flag_plus_14:=FALSE;
END_IF
IF Turbo_Flag_plus_15 THEN
	FOR i:=1 TO 16 DO
		Buffer[15,i].a:=Buffer[15,i].a+Change_volume;
	END_FOR
	Turbo_Flag_plus_15:=FALSE;
END_IF
IF Turbo_Flag_plus_16 THEN
	FOR i:=1 TO 16 DO
		Buffer[16,i].a:=Buffer[16,i].a+Change_volume;
	END_FOR
	Turbo_Flag_plus_16:=FALSE;
END_IF
END_ACTION

(* POU Ввод данных/Get_Currents, ST *)
PROGRAM Get_Currents
VAR
	s32_Current_Inj1,s32_Current_Inj2,s32_Current_Act        : DINT;
   fb_OutGetCurrent   : FB_x_out_get_current;
	s16_Return   	: INT;
	i,j,k: WORD;
END_VAR
(******************* Контроль протекающего тока через выводы на обыв и короткое замыкание *************************************************************)

(* Контроль тока через газовые инжектора осуществляем только если они включены ( включен блок, имеется HOLD ток и не включен спец режим выключения гащза перед переключением на дизель )*)

IF Flag_ECU_ON AND Inj_PWM_time > 0 AND gq_Relay = TRUE		THEN

	fb_OutGetCurrent(ou16_Channel:=X_OUT_06, os32_Current=>s32_Current_Inj1, os16_Status=>s16_Return);			(* Считываем ток, проходящий через инжектора *)
	fb_OutGetCurrent(ou16_Channel:=X_OUT_07, os32_Current=>s32_Current_Inj2, os16_Status=>s16_Return);

	(* Находится ли ток через инжектор 1 в допустимых пределах ? *)
	IF s32_Current_Inj1>Max_inj_current OR s32_Current_Inj1 < Min_inj_current THEN
		i:=i+1;
	ELSE
		i:=0;
	END_IF

	(* Если ток инжектора 1 выходит задопустимые пределы Max_inj_current_time раз подряд, тогда ошибка *)
	IF i>=Max_inj_current_time THEN
		Err_Inj1:=TRUE;
		i:=Max_inj_current_time;					(* Что бы избежать переполнения и ложного сброса флага *)
	ELSE
		Err_Inj2:=FALSE;
	END_IF

	(* Находится ли ток через инжектор 2 в допустимых пределах ? *)
	IF s32_Current_Inj2>Max_inj_current OR s32_Current_Inj2 < Min_inj_current THEN
		j:=j+1;
	ELSE
		j:=0;
	END_IF

	(* Если ток инжектора 2 выходит задопустимые пределы Max_inj_current_time раз подряд, тогда ошибка *)
	IF j>=Max_inj_current_time THEN
		Err_Inj2:=TRUE;
		j:=Max_inj_current_time;					(* Что бы избежать переполнения и ложного сброса флага *)
	ELSE
		Err_Inj2:=FALSE;
	END_IF
END_IF
END_PROGRAM

(* POU Ввод данных/Get_Reductor_press, ST *)
PROGRAM Get_Reductor_press
VAR
	s16_Return      				:INT;
   fb_InGetValue   				:FB_x_in_get_value;


END_VAR
fb_InGetValue(ou16_Channel:=X_IN_22, os32_Value=>Reductor_press, os16_Status=>s16_Return);

(* Находится ли давление в редукторе в допустимых пределах ? *)

IF Reductor_press < Min_Reductor_press THEN
		Count_min_reductor_press:=Count_min_reductor_press+1;
END_IF

(* Если давление в редукторе выходит задопустимые пределы Reductor_press_time раз подряд, тогда ошибка *)
IF Count_min_reductor_press >= Min_Reductor_press_time THEN
		Err_Reductor_press:=TRUE;
		Count_min_reductor_press:=Min_Reductor_press_time;					(* Что бы избежать переполнения и ложного сброса флага *)
ELSE
		Err_Reductor_press:=FALSE;
END_IF
END_PROGRAM

(* POU Act_control, ST *)
PROGRAM Act_control
VAR
	stat: STATISTICS_INT;
	x,y,z: BYTE;  (* Временные переменные, для определения ячейки калибровочной таблицы *)
	Res_stat_pps: BOOL;
	delta:DINT;
	s16_Return      : INT;
   fb_InGetValue   : FB_x_in_get_value;
	i: REAL;


	Flag_PPS_minus: BOOL;
	Flag_PPS_plus: BOOL;
END_VAR
(* Выбираем из калибровочной таблицы занчение желаемой подачи газа, соответствующее текущим оборотам, нагрузке и нажатию на педаль газа*)
fb_InGetValue(ou16_Channel:=X_IN_24, os32_Value=>PPS1, os16_Status=>s16_Return);
fb_InGetValue(ou16_Channel:=X_IN_25, os32_Value=>PPS2, os16_Status=>s16_Return);

IF PPS1 < PPS1_min OR PPS1 > PPS1_max THEN
		Err_PPS:=TRUE;
ELSE
		Err_PPS:=FALSE;
END_IF

IF PPS2 < PPS2_min OR PPS2 > PPS2_max THEN
		Err_PPS:=TRUE;
ELSE
		Err_PPS:=FALSE;
END_IF

i:=PPS1/PPS2;

IF i<0.8 AND i>1.2 THEN
		Err_PPS:=TRUE;
ELSE
		Err_PPS:=FALSE;
END_IF

x:=Get_TURBO_ARRAY_Number(Turbo_pressure);
y:=Get_RPM_ARRAY_Number(RPM);
z:=Get_PPS_ARRAY_Number(PPS1);

(*******************************  Обработка режима эмуляции педали газа **********************************************************)

(* Устанавливаем уровень эмулированности педали газа согласно таблице эмуляции*)
PPS1_emul:= PPS1 - p.PPS_volume[Get_ePPS_ARRAY_Number(PPS1)];

(* Проверка что включен режим dyn=Динамика. Этот режим подразумевает, динамическое
 изменение глубины эмуляции в зависимости от резкости нажатия на педаль 
*) 
IF Flag_PPS_dyn_enable THEN
	delta:=pps1-old_pps;
	IF delta >=0 THEN
		IF delta<150 THEN
			z:=z+1;
			PPS1_emul:=PPS1_emul-100;
			Flag_PPS_plus:=TRUE; (* Флаг показывающий, что глубина эмуляции увеличина *)
		ELSE
			Flag_PPS_plus:=FALSE;
		END_IF

		IF delta>350 THEN
			z:=z+1;
			PPS1_emul:=PPS1_emul+100;
			Flag_PPS_minus:=TRUE; (* Флаг показывающий, что глубина эмуляции уменьшена *)

		ELSE
			Flag_PPS_minus:=FALSE;
		END_IF
	END_IF
Old_pps:=PPS1;
END_IF

(* Установка длительности выдачи газа *)
Inj_PWM_time:=p.Cal_table[ x,y,z ]*4;	(* Переводим в циклы по 250 мкс из мс *)

(* Проверка, что бы эмуляция не выходила за границы возможного физического диапазона *)
IF PPS1_emul<PPS1_min THEN
			PPS1_emul:=1070;
END_IF

IF PPS1_emul>PPS1_max THEN
		PPS1_emul:=4200;
END_IF
END_PROGRAM

(* POU Выборка значения из массива/Get_TURBO_ARRAY_Number, ST *)
FUNCTION Get_TURBO_ARRAY_Number : BYTE
VAR_INPUT
	Turbo_now:DINT;
END_VAR
VAR
	i:BYTE:=1;
	j:BYTE:=16;
	med:BYTE;
END_VAR
(* Функция в качестве аргумента принимает, давление надува в мВольтах, а возвращает номер элемента массива, соответствующего этому количеству оборотов *)


(* Делим массив каждый раз пополам, проверяя где находится искомый элемент, пока границы массива не сойдутся*)

WHILE i<>j  DO
	med:=(i+j)/2;
	IF TURBO_now>p.TURBO_table[med] THEN
		i:=med+1;
	ELSE
		j:=med;
	END_IF
END_WHILE


Get_TURBO_ARRAY_Number :=i;							(* Номер , когда границы сошлись и совпадают с краями массива не нуждается в уточнении *)

(* Уточняем какой элемент массива наиболее сответствует, кол-ву оборотов переданному как элемент функции *)
(* определяем спава или слева от найдено индекса находится ребуемый элемент и в зависмимости от этого действеум *)

IF i=med AND i<>1 THEN
	IF ABS(p.TURBO_table[med-1]-TURBO_now)<= ABS(p.TURBO_table[med]-TURBO_now) THEN
		Get_TURBO_ARRAY_Number :=med-1;
	ELSE
		Get_TURBO_ARRAY_Number :=med;
	END_IF
ELSIF i<>med AND  i<>16 THEN
	IF ABS(p.TURBO_table[med+1]-TURBO_now)<= ABS(p.TURBO_table[med]-TURBO_now) THEN
		Get_TURBO_ARRAY_Number :=med+1;
	ELSE
		Get_TURBO_ARRAY_Number :=med;
	END_IF
END_IF
END_FUNCTION

(* POU Выборка значения из массива/Get_RPM_ARRAY_Number, ST *)
FUNCTION Get_RPM_ARRAY_Number : BYTE
VAR_INPUT
	RPM_now:DINT;
END_VAR
VAR
	i:BYTE:=1;
	j:BYTE:=16;
	med:BYTE;
END_VAR
(* Функция в качестве аргумента принимает, количество оборотов, а возвращает номер элемента массива, соответствующего этому количеству оборотов *)


(* Делим массив каждый раз пополам, проверяя где находится искомый элемент, пока границы массива не сойдутся*)

WHILE i<>j  DO
	med:=(i+j)/2;
	IF RPM_now>p.RPM_table[med] THEN
		i:=med+1;
	ELSE
		j:=med;
	END_IF
END_WHILE


Get_RPM_ARRAY_Number :=i;							(* Номер , когда границы сошлись и совпадают с краями массива не нуждается в уточнении *)

(* Уточняем какой элемент массива наиболее сответствует, кол-ву оборотов переданному как элемент функции *)
(* определяем спава или слева от найдено индекса находится ребуемый элемент и в зависмимости от этого действеум *)

IF i=med AND i<>1 THEN
	IF ABS(p.RPM_table[med-1]-RPM_now)<= ABS(p.RPM_table[med]-RPM_now) THEN
		Get_RPM_ARRAY_Number :=med-1;
	ELSE
		Get_RPM_ARRAY_Number :=med;
	END_IF
ELSIF i<>med AND  i<>16 THEN
	IF ABS(p.RPM_table[med+1]-RPM_now)<= ABS(p.RPM_table[med]-RPM_now) THEN
		Get_RPM_ARRAY_Number :=med+1;
	ELSE
		Get_RPM_ARRAY_Number :=med;
	END_IF
END_IF
END_FUNCTION

(* POU Выборка значения из массива/Get_PPS_ARRAY_Number, ST *)
FUNCTION Get_PPS_ARRAY_Number : BYTE
VAR_INPUT
	PPS_now:DINT;
END_VAR
VAR
	i:BYTE:=1;
	j:BYTE:=16;
	med:BYTE;
END_VAR
(* Функция в качестве аргумента принимает, количество оборотов, а возвращает номер элемента массива, соответствующего этому PPS *)


(* Делим массив каждый раз пополам, проверяя где находится искомый элемент, пока границы массива не сойдутся*)

WHILE i<>j  DO
	med:=(i+j)/2;
	IF PPS_now>p.PPS_table[med] THEN
		i:=med+1;
	ELSE
		j:=med;
	END_IF
END_WHILE


Get_PPS_ARRAY_Number :=i;							(* Номер , когда границы сошлись и совпадают с краями массива не нуждается в уточнении *)

(* Уточняем какой элемент массива наиболее сответствует, кол-ву оборотов переданному как элемент функции *)
(* определяем спава или слева от найдено индекса находится ребуемый элемент и в зависмимости от этого действеум *)

IF i=med AND i<>1 THEN
	IF ABS(p.PPS_table[med-1]-PPS_now)<= ABS(p.RPM_table[med]-PPS_now) THEN
		Get_PPS_ARRAY_Number :=med-1;
	ELSE
		Get_PPS_ARRAY_Number :=med;
	END_IF
ELSIF i<>med AND  i<>16 THEN
	IF ABS(p.PPS_table[med+1]-PPS_now)<= ABS(p.PPS_table[med]-PPS_now) THEN
		Get_PPS_ARRAY_Number :=med+1;
	ELSE
		Get_PPS_ARRAY_Number :=med;
	END_IF
END_IF
END_FUNCTION

(* POU Выборка значения из массива/Get_ePPS_ARRAY_Number, ST *)
FUNCTION Get_ePPS_ARRAY_Number : BYTE
VAR_INPUT
	PPS_now:DINT;
END_VAR
VAR
	i:BYTE:=1;
	j:BYTE:=32;
	med:BYTE;
END_VAR
(* Функция в качестве аргумента принимает, количество оборотов, а возвращает номер элемента массива, соответствующего этому количеству оборотов *)


(* Делим массив каждый раз пополам, проверяя где находится искомый элемент, пока границы массива не сойдутся*)

WHILE i<>j  DO
	med:=(i+j)/2;
	IF PPS_now>p.PPS_index[med] THEN
		i:=med+1;
	ELSE
		j:=med;
	END_IF
END_WHILE


Get_ePPS_ARRAY_Number :=i;							(* Номер , когда границы сошлись и совпадают с краями массива не нуждается в уточнении *)

(* Уточняем какой элемент массива наиболее сответствует, кол-ву оборотов переданному как элемент функции *)
(* определяем спава или слева от найдено индекса находится ребуемый элемент и в зависмимости от этого действеум *)

IF i=med AND i<>1 THEN
	IF ABS(p.PPS_index[med-1]-PPS_now)<= ABS(p.PPS_index[med]-PPS_now) THEN
		Get_ePPS_ARRAY_Number :=med-1;
	ELSE
		Get_ePPS_ARRAY_Number :=med;
	END_IF
ELSIF i<>med AND  i<>16 THEN
	IF ABS(p.PPS_index[med+1]-PPS_now)<= ABS(p.PPS_index[med]-PPS_now) THEN
		Get_ePPS_ARRAY_Number :=med+1;
	ELSE
		Get_ePPS_ARRAY_Number :=med;
	END_IF
END_IF
END_FUNCTION

(* POU Ввод данных/Get_Turbo_EGR, ST *)
PROGRAM Get_Turbo_EGR
VAR
	s16_Return      : INT;
   fb_InGetValue   : FB_x_in_get_value;
END_VAR
fb_InGetValue(ou16_Channel:=X_IN_21, os32_Value=>Turbo_pressure, os16_Status=>s16_Return);
fb_InGetValue(ou16_Channel:=X_IN_14, os32_Value=>EGR, os16_Status=>s16_Return);
END_PROGRAM

(* POU Ввод данных/Get_Key, ST *)
PROGRAM Get_Key
VAR
	s16_Return      : INT;
   fb_InGetValue   : FB_x_in_get_value;

	DF_switch	:DINT;
	DF_flag		:BOOL;

END_VAR
fb_InGetValue(ou16_Channel:=X_IN_12, os32_Value=>DF_switch, os16_Status=>s16_Return);

IF DF_switch=0 THEN					(* Если конпока изменения режима работы ECU нажата, то...*)
	IF DF_flag THEN					(* Первый ли цикл когда она нажата ? *)
		DF_flag:=FALSE;				(*Выставляем флажок, для  игнорирования этой ветви, до тех пор пока кнопка не изменит своего положения *)
		IF Flag_ECU_ON THEN			(* Включаем или выключаем газодизельный режим ECU*)
			Flag_ECU_ON:=FALSE;
		ELSE
			Flag_ECU_ON:=TRUE;
			Count_min_reductor_press:=0; (* При переключении режимов начать отчет времени когда далвение было минимальным с 0 *)
		END_IF;
	END_IF
ELSE
	DF_flag:=TRUE;				(* Кнопка была отпущена, устанвкливаем разрешительный флажок для обработки следующего нажатия *)
END_IF
END_PROGRAM

(* POU Put_emul, ST *)
PROGRAM Put_emul
VAR
	i,j						:DINT;

	s16_Return           :INT;
	fb_OutSetValue   : FB_x_out_set_value;
END_VAR
(* Если не включен режим исследования зависимости PWM и выхода напряжения с операционного усилителя, то выдаем значения PWM из таблицы соответствия PWM напряжению *)

IF Flag_PWM_researh=FALSE THEN
	(* Выборка уровня PWM для выдачи на операционный усилитель для емуляции PPS1 *)
	CASE PPS1_emul OF
			0..900:		 	j:=p.PPS1_emul_PWM[1];
			901..1000:		j:=p.PPS1_emul_PWM[2];
			1001..1100:		j:=p.PPS1_emul_PWM[3];
			1101..1200:		j:=p.PPS1_emul_PWM[4];
			1201..1300:		j:=p.PPS1_emul_PWM[5];
			1301..1400:		j:=p.PPS1_emul_PWM[6];
			1401..1500: 	j:=p.PPS1_emul_PWM[7];
			1501..1600:		j:=p.PPS1_emul_PWM[8];
			1601..1700:		j:=p.PPS1_emul_PWM[9];
			1701..1800: 	j:=p.PPS1_emul_PWM[10];
			1801..1900:		j:=p.PPS1_emul_PWM[11];
			1901..2000:		j:=p.PPS1_emul_PWM[12];
			2001..2100: 	j:=p.PPS1_emul_PWM[13];
			2101..2200:		j:=p.PPS1_emul_PWM[14];
			2201..2300:		j:=p.PPS1_emul_PWM[15];
			2301..2400: 	j:=p.PPS1_emul_PWM[16];
			2401..2500:		j:=p.PPS1_emul_PWM[17];
			2501..2600:		j:=p.PPS1_emul_PWM[18];
			2601..2700: 	j:=p.PPS1_emul_PWM[19];
			2701..2800:		j:=p.PPS1_emul_PWM[20];
			2801..2900:		j:=p.PPS1_emul_PWM[21];
			2901..3000: 	j:=p.PPS1_emul_PWM[22];
			3001..3100:		j:=p.PPS1_emul_PWM[23];
			3101..3200:		j:=p.PPS1_emul_PWM[24];
			3201..3300: 	j:=p.PPS1_emul_PWM[25];
			3301..3400:		j:=p.PPS1_emul_PWM[26];
			3401..3500:		j:=p.PPS1_emul_PWM[27];
			3501..3600: 	j:=p.PPS1_emul_PWM[28];
			3601..3700:		j:=p.PPS1_emul_PWM[29];
			3701..3800: 	j:=p.PPS1_emul_PWM[30];
			3801..3900:		j:=p.PPS1_emul_PWM[31];
			3901..4000:		j:=p.PPS1_emul_PWM[32];
			4001..4100: 	j:=p.PPS1_emul_PWM[33];
			4101..4200:		j:=p.PPS1_emul_PWM[34];
			4201..5000:		j:=p.PPS1_emul_PWM[35];
	END_CASE

END_IF

(* ePPS1 *)
fb_OutSetValue(ou16_Channel:=X_OUT_08, os32_Value:=j, os16_Status=>s16_Return);
END_PROGRAM

(* POU Ввод данных/Get_EGT, ST *)
PROGRAM Get_EGT
VAR
	s16_Return      : INT;
   fb_InGetValue   : FB_x_in_get_value;

	EGT_err_flag: BOOL;
	Count_max_EGT: WORD;
	Flag_EGT_reset: BOOL;
END_VAR
fb_InGetValue(ou16_Channel:=X_IN_23, os32_Value=>EGT, os16_Status=>s16_Return);

(* Если EGT превысило допустимую температуру, то следующий контроль EGT на возможное включение блока произойдет через некоторое время *)

IF EGT_err_flag AND  Count_max_EGT < EGT_err_time THEN
	Count_max_EGT:=Count_max_EGT+1;
ELSE
	Count_max_EGT:=0;
	(* Находится ли EGT в допустимых пределах ? *)
	IF EGT>=p.EGT_max THEN
		EGT_err_flag:=TRUE;
		Err_EGT:=TRUE;
	ELSE
		EGT_err_flag:=FALSE;
		Err_EGT:=FALSE;
	END_IF
END_IF

(* Контроль, что бы между сменами режимов прошло достаточно кол-ва времени *)
IF (gu32_TimeMs-Turn_start) > Min_time_cnange_mode_EGT THEN
(* Запись максимального значения EGT в как течении сесии так и абсолютно за все время *)
		IF Flag_ECU_ON THEN
				IF EGT > a.EGT_max_sessions_GAS	THEN
					a.EGT_max_sessions_GAS:=EGT;
				END_IF
				IF EGT > a.EGT_max_abs_GAS	THEN
					a.EGT_max_abs_GAS:=EGT;
				END_IF
		ELSE
				IF EGT > a.EGT_max_sessions_DIESEL	THEN
					a.EGT_max_sessions_DIESEL:=EGT;
				END_IF
				IF EGT > a.EGT_max_abs_DIESEL	THEN
					a.EGT_max_abs_DIESEL:=EGT;
				END_IF
		END_IF
END_IF

IF Flag_EGT_reset THEN
	a.Flag_byte:=128+64;
	a.EGT_max_abs_GAS:=0;
	a.EGT_max_abs_DIESEL:=0;
	a.EGT_max_sessions_GAS:=0;
	a.EGT_max_sessions_DIESEL:=0;
	Flag_EGT_reset:=FALSE;
END_IF
END_PROGRAM

(* POU Ввод данных/Get_Gas_meter, ST *)
PROGRAM Get_Gas_meter
VAR
	s16_Return      : INT;
   fb_InGetValue   : FB_x_in_get_value;
	fb_OutSetValue   : FB_x_out_set_value;

	i: DINT;
END_VAR
(* Считать значениедатчика кол-ва газа *)
fb_InGetValue(ou16_Channel:=X_IN_02, os32_Value=>Gas_meter, os16_Status=>s16_Return);
(* Определить уровень PWM для зажигания LED *)
i:=p.LED_BAR_PWM[Get_Gas_meter_ARRAY_Number(Gas_meter)];

(* Выдать PWM на LED bar *)
fb_OutSetValue(ou16_Channel:=X_OUT_03, os32_Value:=i, os16_Status=>s16_Return);
END_PROGRAM

(* POU Выборка значения из массива/Get_Gas_meter_ARRAY_Number, ST *)
FUNCTION Get_Gas_meter_ARRAY_Number : BYTE
VAR_INPUT
	Gas_meter_now:DINT;
END_VAR
VAR
	i:BYTE:=1;
	j:BYTE:=5;
	med:BYTE;
	Gas_meter_volume: BOOL;
END_VAR
(* Функция в качестве аргумента принимает, количество оборотов, а возвращает номер элемента массива, соответствующего этому PPS *)


(* Делим массив каждый раз пополам, проверяя где находится искомый элемент, пока границы массива не сойдутся*)

WHILE i<>j  DO
	med:=(i+j)/2;
	IF Gas_meter_now>p.Gas_meter_volume[med] THEN
		i:=med+1;
	ELSE
		j:=med;
	END_IF
END_WHILE


Get_Gas_meter_ARRAY_Number :=i;							(* Номер , когда границы сошлись и совпадают с краями массива не нуждается в уточнении *)

(* Уточняем какой элемент массива наиболее сответствует, кол-ву оборотов переданному как элемент функции *)
(* определяем спава или слева от найдено индекса находится ребуемый элемент и в зависмимости от этого действеум *)

IF i=med AND i<>1 THEN
	IF ABS(p.Gas_meter_volume[med-1]-Gas_meter_now)<= ABS(p.Gas_meter_volume[med]-Gas_meter_now) THEN
		Get_Gas_meter_ARRAY_Number :=med-1;
	ELSE
		Get_Gas_meter_ARRAY_Number :=med;
	END_IF
ELSIF i<>med AND  i<>16 THEN
	IF ABS(p.Gas_meter_volume[med+1]-Gas_meter_now)<= ABS(p.Gas_meter_volume[med]-Gas_meter_now) THEN
		Get_Gas_meter_ARRAY_Number :=med+1;
	ELSE
		Get_Gas_meter_ARRAY_Number :=med;
	END_IF
END_IF
END_FUNCTION

(* POU Ввод данных/Get_Reductor_temp, ST *)
PROGRAM Get_Reductor_temp
VAR
	s16_Return      : INT;
   fb_InGetValue   : FB_x_in_get_value;
END_VAR
fb_InGetValue(ou16_Channel:=X_IN_20, os32_Value=>Reductor_temp, os16_Status=>s16_Return);

IF Reductor_temp<Reductor_temp_work THEN
	Err_Reductor_temp:=TRUE;
ELSE
	Err_Reductor_temp:=FALSE;
END_IF
END_PROGRAM

(* POU Ввод данных/Get_Inj_temp, ST *)
PROGRAM Get_Inj_temp
VAR
	s16_Return      : INT;
   fb_InGetValue   : FB_x_in_get_value;
END_VAR
fb_InGetValue(ou16_Channel:=X_IN_15, os32_Value=>Injector_temp, os16_Status=>s16_Return);

(* Находится ли температура форсунок в допустимых пределах ? *)
(* Если температура форсунок хоть один раз превысила допустимый порог, то снять ошибку можно только перегрузкой *)

IF Injector_temp > Inj_temp_max THEN
	Err_inj_temp:=TRUE;
END_IF
END_PROGRAM

(* POU CAN/Send, ST *)
PROGRAM Send
VAR
	s16_Return       		: INT;
	t_Msg             	: T_x_can_msg;
   fb_CanObjSendMsg   	: FB_x_can_obj_send_msg;
	fb_EepRead  			: FB_x_eep_read;
	u16_Crc           	: UINT;
	fb_UtiCalcCrc16   	: FB_x_uti_calc_crc_16;
	CAN_TX_count			:WORD:=10000;				(* Счетчик переданных пакетов по CAN *)

END_VAR
IF Flag_CAN THEN

	IF Flag_CAN_Write THEN
		Flag_CAN_Write:=FALSE;
		t_Msg.t_Id.u32_Id := 16#101;
		t_Msg.t_Id.u8_Xtd := 0;
		t_Msg.u8_Dlc      := 8;				(* Количество передаваемых байт *)
		t_Msg.au8_Data[0] := 1;
		t_Msg.au8_Data[1] := 9;
		t_Msg.au8_Data[2] := 7;
		t_Msg.au8_Data[3] := 2;
		t_Msg.au8_Data[4] := 1;
		t_Msg.au8_Data[5] := 9;
		t_Msg.au8_Data[6] := 7;
		t_Msg.au8_Data[7] := 2;
		fb_CanObjSendMsg(ou32_Handle:=TX, ot_Msg:=t_Msg, os16_Status=>s16_Return);
	END_IF


	IF Flag_CAN_send THEN											(* Первоначальная процедура, выполняется один раз по команде от Питоновской программе *)
		(* Читаем все содержимое энергонезависимой памяти *)
		fb_EepRead(ou32_Address:=0, ou32_Count:=SIZEOF(Can_buffer), opu8_Data:=ADR(Can_buffer), os16_Status=>s16_Return);
		(* Вычисляем CRC16 для массива передаваемых данных *)
		u16_Crc:=16#1D0F;
		fb_UtiCalcCrc16(ou32_Count:=SIZEOF(Can_buffer)-2, opu8_Data:=ADR(Can_buffer), ou16_Crc:=u16_Crc, os16_Status=>s16_Return);
		Can_buffer[SIZEOF(Can_buffer)-1]:=WORD_TO_BYTE(u16_Crc);
		Can_buffer[SIZEOF(Can_buffer)]:=WORD_TO_BYTE(u16_Crc/256);
		CAN_TX_count:=0;
		Flag_CAN_send:=FALSE;


	ELSIF CAN_TX_count <=  (SIZEOF(Can_buffer)-8) THEN						(* Передача основных данных, выполняется 1 раз после хандшейка *)

			(* Постоянная часть передачи *)
			t_Msg.t_Id.u32_Id := 16#101;		(* Адрес пакета *)
			t_Msg.t_Id.u8_Xtd := 0;
			t_Msg.u8_Dlc      := 8;				(* Количество передаваемых байт *)
			t_Msg.au8_Data[0] := Can_buffer[CAN_TX_count+1];
			t_Msg.au8_Data[1] := Can_buffer[CAN_TX_count+2];
			t_Msg.au8_Data[2] := Can_buffer[CAN_TX_count+3];
			t_Msg.au8_Data[3] := Can_buffer[CAN_TX_count+4];
			t_Msg.au8_Data[4] := Can_buffer[CAN_TX_count+5];
			t_Msg.au8_Data[5] := Can_buffer[CAN_TX_count+6];
			t_Msg.au8_Data[6] := Can_buffer[CAN_TX_count+7];
			t_Msg.au8_Data[7] := Can_buffer[CAN_TX_count+8];
			fb_CanObjSendMsg(ou32_Handle:=TX, ot_Msg:=t_Msg, os16_Status=>s16_Return);
			CAN_TX_count:=CAN_TX_count+8;
		END_IF

END_IF
END_PROGRAM

(* POU CAN/Recieve, ST *)
PROGRAM Recieve
VAR
	s16_Return        	: INT;
	r_Msg			         : T_x_can_msg;
	fb_CanObjGetMsg   	: FB_x_can_obj_get_msg;
	fb_EepWrite  			: FB_x_eep_write;

	u16_Crc           	: UINT;
	fb_UtiCalcCrc16   	: FB_x_uti_calc_crc_16;
	i: WORD; (* Счетчик принятых по CAN пакетов в калибровке *)

	crc_given: UINT;
END_VAR
IF Flag_CAN THEN
			(* Что бы при ошибке чтения с CANa , при не изменении значений не произошо ложного срабатывания *)
			r_Msg.au8_Data[0]:=0;r_Msg.au8_Data[1]:=0;r_Msg.au8_Data[2]:=0;r_Msg.au8_Data[3]:=0;r_Msg.au8_Data[4]:=0;
			r_Msg.au8_Data[5]:=0;r_Msg.au8_Data[6]:=0;r_Msg.au8_Data[7]:=0;
			fb_CanObjGetMsg(ou32_Handle:=RX, ot_Msg=>r_Msg, os16_Status=>s16_Return);
			IF s16_Return = C_NO_ERR THEN

					(* Поступил запрос на передачу? *)
					IF	Flag_CAN_recieve=FALSE AND r_Msg.au8_Data[0] = 8 AND r_Msg.au8_Data[1] = 7 AND r_Msg.au8_Data[2] = 6 AND r_Msg.au8_Data[3] = 5 AND
						r_Msg.au8_Data[4] = 4 AND r_Msg.au8_Data[5] = 3 AND r_Msg.au8_Data[6] = 2 AND	r_Msg.au8_Data[7] = 1 THEN
						Flag_CAN_send:=TRUE;
					END_IF

					(* Поступил запрос на прием ? *)
					IF Flag_CAN_recieve = FALSE AND r_Msg.au8_Data[0] = 1 AND r_Msg.au8_Data[1] = 2 AND r_Msg.au8_Data[2] = 3 AND r_Msg.au8_Data[3] = 4 AND
						r_Msg.au8_Data[4] = 5 AND r_Msg.au8_Data[5] = 6 AND r_Msg.au8_Data[6] = 7 AND r_Msg.au8_Data[7] = 8 THEN

									Flag_CAN_recieve:=TRUE;
									i:=1;
					ELSIF i <= SIZEOF(Can_buffer)-7 THEN
											Can_buffer[i]:=r_Msg.au8_Data[0]; Can_buffer[i+1]:=r_Msg.au8_Data[1]; Can_buffer[i+2]:=r_Msg.au8_Data[2]; Can_buffer[i+3]:=r_Msg.au8_Data[3];
											Can_buffer[i+4]:=r_Msg.au8_Data[4]; Can_buffer[i+5]:=r_Msg.au8_Data[5]; Can_buffer[i+6]:=r_Msg.au8_Data[6]; Can_buffer[i+7]:=r_Msg.au8_Data[7];
											i:=i+8;
											IF i=SIZEOF(Can_buffer)+1 THEN
													Flag_CAN_recieve:= FALSE;
													(* Вычисляем CRC16 для массива передаваемых данных *)
													u16_Crc:=16#1D0F;
													fb_UtiCalcCrc16(ou32_Count:=SIZEOF(Can_buffer)-2, opu8_Data:=ADR(Can_buffer), ou16_Crc:=u16_Crc, os16_Status=>s16_Return);
													crc_given:= Can_buffer[SIZEOF(Can_buffer)]*256+Can_buffer[SIZEOF(Can_buffer)-1];
													IF crc_given =  u16_Crc THEN
															fb_EepWrite(ou32_Address:=0, ou32_Count:=SIZEOF(Can_buffer), opu8_Data:=ADR(Can_buffer), os16_Status=>s16_Return);
															Flag_CAN_Write:= TRUE;
													END_IF
											END_IF
					END_IF

			END_IF
END_IF
END_PROGRAM

(* POU Ввод данных/Get_PPS, ST *)
PROGRAM Get_PPS
VAR

END_VAR

END_PROGRAM

(* Visualisation Check_parameters/CHECK_CURRENT
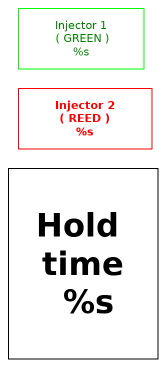
rounded rectangle at (1200,110)-(1326,171): text "Injector 1 / ( GREEN ) / %s"; shows Get_Currents.s32_Current_Inj1/1000
rounded rectangle at (1200,190)-(1334,251): text "Injector 2 / ( REED ) / %s"; shows Get_Currents.s32_Current_Inj2/1000
rounded rectangle at (1190,270)-(1340,461): text "Hold / time / %s"; shows .Inj_PWM_time/4
1 more shapes without text or variables
1 elements of other kinds (tables, trends, ...) not read
*)

(* Visualisation Check_parameters/CHECK_EGT_EGR
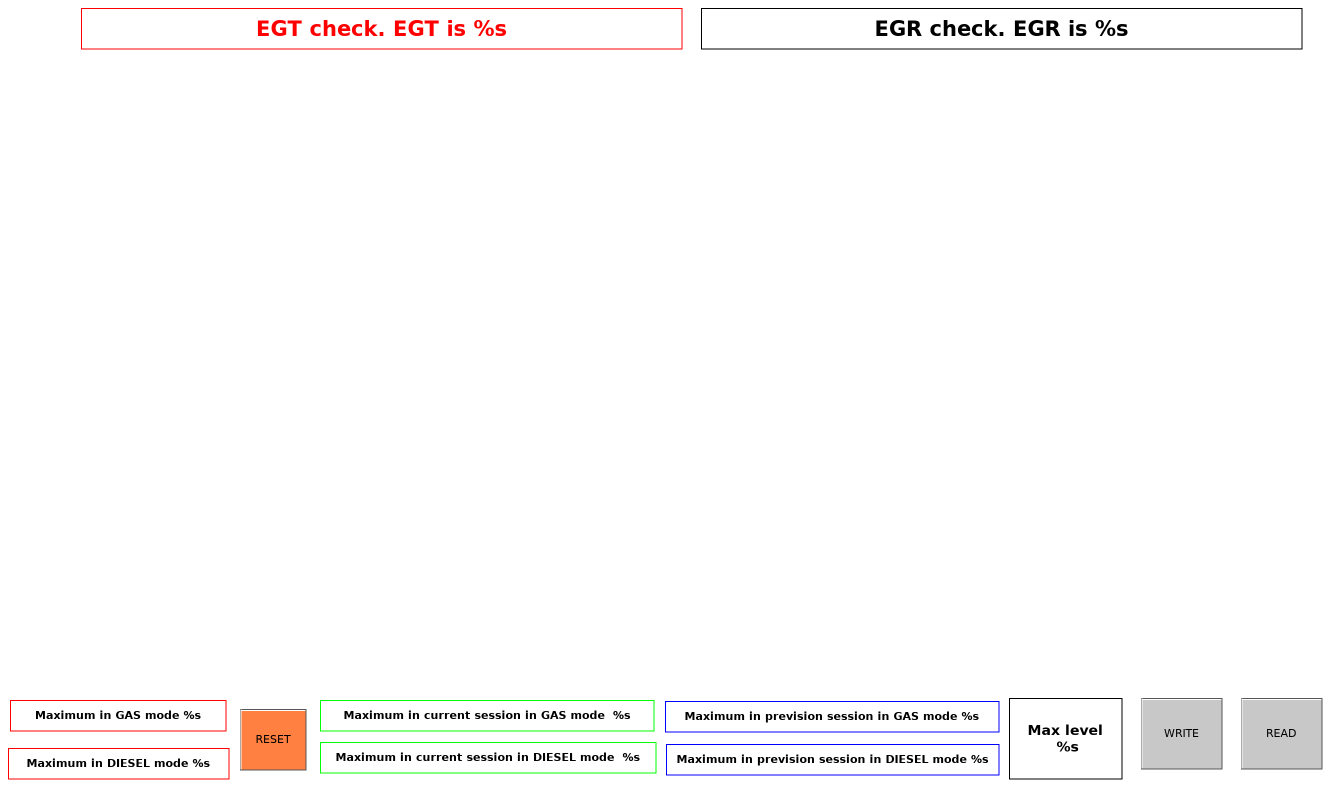
rounded rectangle at (9,702)-(225,733): text "Maximum in GAS mode %s"; shows .a.EGT_max_abs_GAS
rounded rectangle at (7,750)-(228,781): text "Maximum in DIESEL mode %s"; shows .a.EGT_max_abs_DIESEL
rounded rectangle at (665,746)-(998,777): text "Maximum in prevision session in DIESEL mode %s"; shows PLC_PRG.EGT_max_prev_sessions_DIESEL
rounded rectangle at (664,703)-(998,734): text "Maximum in prevision session in GAS mode %s"; shows PLC_PRG.EGT_max_prev_sessions_GAS
rounded rectangle at (319,702)-(653,733): text "Maximum in current session in GAS mode  %s"; shows .a.EGT_max_sessions_GAS
rounded rectangle at (319,744)-(655,775): text "Maximum in current session in DIESEL mode  %s"; shows .a.EGT_max_sessions_DIESEL
rounded rectangle at (80,10)-(681,51): text "EGT check. EGT is %s"; shows .EGT
rounded rectangle at (1008,700)-(1121,781): text "Max level / %s"; shows .p.EGT_max; editable
button at (1240,700)-(1321,771): text "READ"; taps Parameters_read_write.Flag_Parameters_read
button at (1140,700)-(1221,771): text "WRITE"; taps Parameters_read_write.Flag_Parameters_write
button at (239,711)-(305,772): text "RESET"; taps Get_EGT.Flag_EGT_reset
rounded rectangle at (700,10)-(1301,51): text "EGR check. EGR is %s"; shows .EGR
1 elements of other kinds (tables, trends, ...) not read
*)

(* Visualisation Check_parameters/CHECK_INJ_TEMP
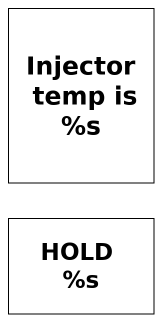
rounded rectangle at (1200,50)-(1346,225): text "Injector / temp is / %s"; shows .Injector_temp
rounded rectangle at (1200,260)-(1346,356): text "HOLD / %s"; shows .Inj_PWM_time/4
1 more shapes without text or variables
1 elements of other kinds (tables, trends, ...) not read
*)

(* Visualisation EMUL_PWM_RESEARCH
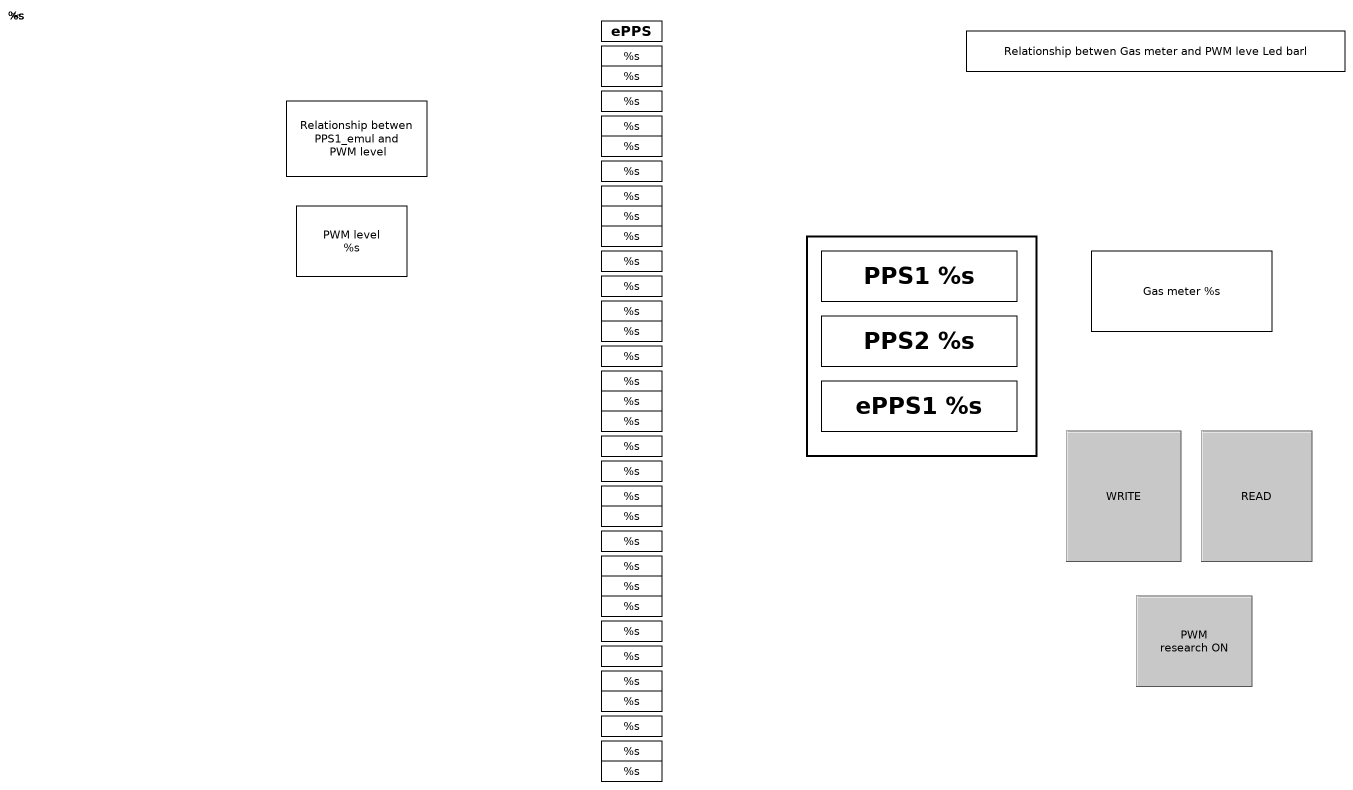
button at (1120,580)-(1236,671): text "PWM / research ON"; toggles .Flag_PWM_researh
button at (1050,415)-(1165,546): text "WRITE"; taps DFPRS_Change_Cal_Table.Write_cal
button at (1185,415)-(1296,546): text "READ"; taps DFPRS_Change_Cal_Table.Read_cal
rounded rectangle at (950,15)-(1329,56): text "Relationship betwen Gas meter and PWM leve Led barl"
rounded rectangle at (1075,235)-(1256,316): text "Gas meter %s"; shows .Gas_meter
rounded rectangle at (270,85)-(411,161): text "Relationship betwen / PPS1_emul and / PWM level"
rectangle at (0,0)-(0,0): text "%s"; shows p.LED_BAR_PWM[INDEX]; editable
rectangle at (0,0)-(0,0): text "%s"; shows p.Gas_meter_volume[INDEX]; editable
rounded rectangle at (280,190)-(391,261): text "PWM level / %s"; shows Put_emul.j; editable
rectangle at (0,0)-(0,0): text "%s"; shows p.PPS1_emul_PWM[INDEX]; editable
rectangle at (0,0)-(0,0): text "%s"; shows p.PPS_index[INDEX]; editable
rectangle at (0,0)-(0,0): text "%s"; shows p.PPS_volume[INDEX]; editable
rounded rectangle at (805,235)-(1001,286): text "PPS1 %s"; shows .PPS1
rounded rectangle at (805,300)-(1001,351): text "PPS2 %s"; shows .PPS2
rounded rectangle at (805,365)-(1001,416): text "ePPS1 %s"; shows .PPS1_emul
rectangle at (0,0)-(0,0): text "%s"; shows p.PPS1_emul_PWM_U[INDEX]; editable
rectangle at (585,30)-(646,51): text "%s"; shows p.PPS_index[1]-p.PPS_volume[1]
rectangle at (585,50)-(646,71): text "%s"; shows p.PPS_index[2]-p.PPS_volume[2]
rectangle at (585,75)-(646,96): text "%s"; shows p.PPS_index[3]-p.PPS_volume[3]
rectangle at (585,100)-(646,121): text "%s"; shows p.PPS_index[4]-p.PPS_volume[4]
rectangle at (585,120)-(646,141): text "%s"; shows p.PPS_index[5]-p.PPS_volume[5]
rectangle at (585,145)-(646,166): text "%s"; shows p.PPS_index[6]-p.PPS_volume[6]
rectangle at (585,170)-(646,191): text "%s"; shows p.PPS_index[7]-p.PPS_volume[7]
rectangle at (585,190)-(646,211): text "%s"; shows p.PPS_index[8]-p.PPS_volume[8]
rectangle at (585,210)-(646,231): text "%s"; shows p.PPS_index[9]-p.PPS_volume[9]
rectangle at (585,235)-(646,256): text "%s"; shows p.PPS_index[10]-p.PPS_volume[10]
rectangle at (585,260)-(646,281): text "%s"; shows p.PPS_index[11]-p.PPS_volume[11]
rectangle at (585,285)-(646,306): text "%s"; shows p.PPS_index[12]-p.PPS_volume[12]
rectangle at (585,305)-(646,326): text "%s"; shows p.PPS_index[13]-p.PPS_volume[13]
rectangle at (585,330)-(646,351): text "%s"; shows p.PPS_index[14]-p.PPS_volume[14]
rectangle at (585,355)-(646,376): text "%s"; shows p.PPS_index[15]-p.PPS_volume[15]
rectangle at (585,375)-(646,396): text "%s"; shows p.PPS_index[16]-p.PPS_volume[16]
rectangle at (585,395)-(646,416): text "%s"; shows p.PPS_index[17]-p.PPS_volume[17]
rectangle at (585,420)-(646,441): text "%s"; shows p.PPS_index[18]-p.PPS_volume[18]
rectangle at (585,445)-(646,466): text "%s"; shows p.PPS_index[19]-p.PPS_volume[19]
rectangle at (585,470)-(646,491): text "%s"; shows p.PPS_index[20]-p.PPS_volume[20]
rectangle at (585,490)-(646,511): text "%s"; shows p.PPS_index[21]-p.PPS_volume[21]
rectangle at (585,515)-(646,536): text "%s"; shows p.PPS_index[22]-p.PPS_volume[22]
rectangle at (585,540)-(646,561): text "%s"; shows p.PPS_index[23]-p.PPS_volume[23]
rectangle at (585,560)-(646,581): text "%s"; shows p.PPS_index[24]-p.PPS_volume[24]
rectangle at (585,580)-(646,601): text "%s"; shows p.PPS_index[25]-p.PPS_volume[25]
rectangle at (585,605)-(646,626): text "%s"; shows p.PPS_index[26]-p.PPS_volume[26]
rectangle at (585,630)-(646,651): text "%s"; shows p.PPS_index[27]-p.PPS_volume[27]
rectangle at (585,655)-(646,676): text "%s"; shows p.PPS_index[28]-p.PPS_volume[28]
rectangle at (585,675)-(646,696): text "%s"; shows p.PPS_index[29]-p.PPS_volume[29]
rectangle at (585,700)-(646,721): text "%s"; shows p.PPS_index[30]-p.PPS_volume[30]
rectangle at (585,725)-(646,746): text "%s"; shows p.PPS_index[31]-p.PPS_volume[31]
rectangle at (585,745)-(646,766): text "%s"; shows p.PPS_index[32]-p.PPS_volume[32]
rectangle at (585,5)-(646,26): text "ePPS"
1 more shapes without text or variables
*)

(* Visualisation GAS_CALIBRATION
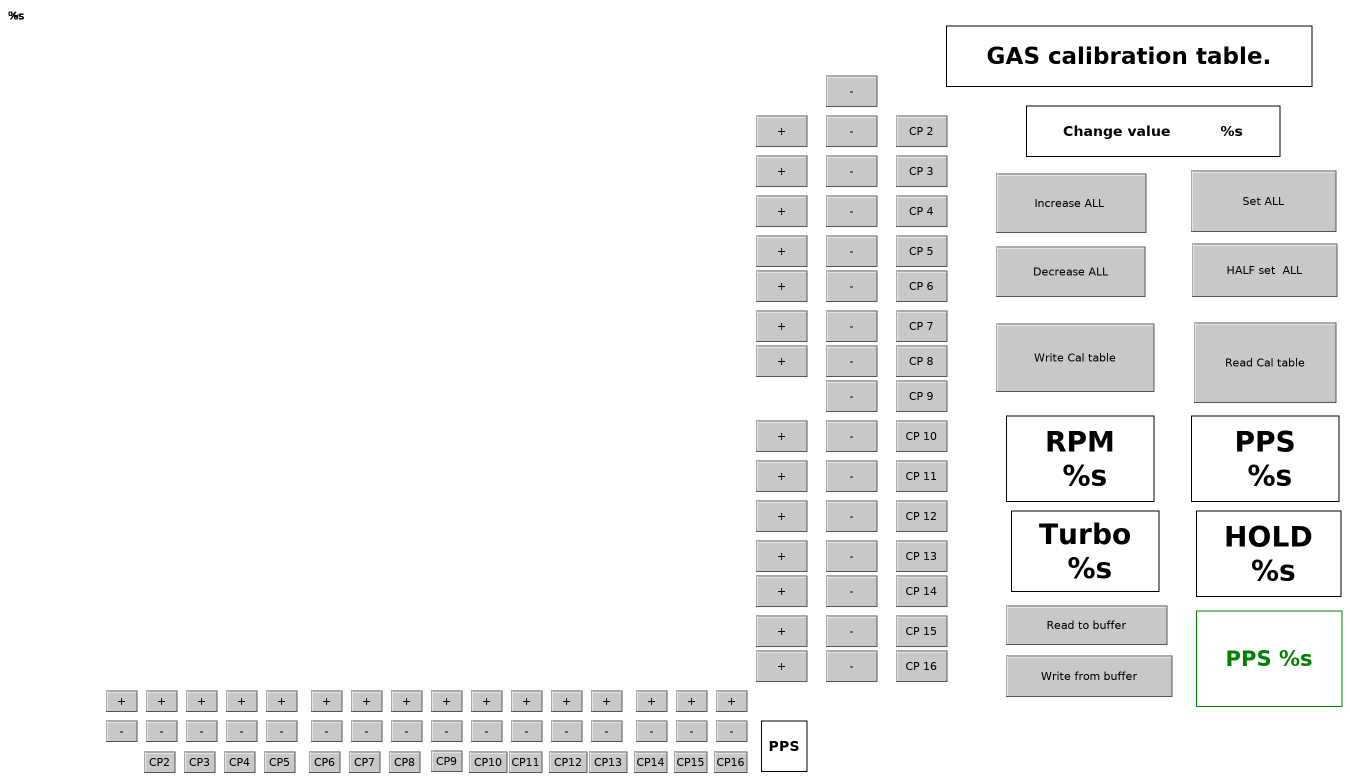
rectangle at (0,0)-(0,0): text "%s"; shows p.RPM_table[INDEX]; editable
rectangle at (0,0)-(0,0): text "%s"; shows p.Turbo_table[1]; editable
rectangle at (0,0)-(0,0): text "%s"; shows p.Turbo_table[2]; editable
rectangle at (0,0)-(0,0): text "%s"; shows p.Turbo_table[3]; editable
rectangle at (0,0)-(0,0): text "%s"; shows p.Turbo_table[4]; editable
rectangle at (0,0)-(0,0): text "%s"; shows p.Turbo_table[5]; editable
rectangle at (0,0)-(0,0): text "%s"; shows p.Turbo_table[6]; editable
rectangle at (0,0)-(0,0): text "%s"; shows p.Turbo_table[7]; editable
rectangle at (0,0)-(0,0): text "%s"; shows p.Turbo_table[8]; editable
rectangle at (0,0)-(0,0): text "%s"; shows p.Turbo_table[9]; editable
rectangle at (0,0)-(0,0): text "%s"; shows p.Turbo_table[10]; editable
rectangle at (0,0)-(0,0): text "%s"; shows p.Turbo_table[11]; editable
rectangle at (0,0)-(0,0): text "%s"; shows p.Turbo_table[12]; editable
rectangle at (0,0)-(0,0): text "%s"; shows p.Turbo_table[13]; editable
rectangle at (0,0)-(0,0): text "%s"; shows p.Turbo_table[14]; editable
rectangle at (0,0)-(0,0): text "%s"; shows p.Turbo_table[15]; editable
rectangle at (0,0)-(0,0): text "%s"; shows p.Turbo_table[16]; editable
rounded rectangle at (1180,595)-(1326,691): text "PPS %s"; shows DFPRS_Change_Cal_Table.PPS_number; editable
button at (980,158)-(1130,217): text "Increase ALL"; taps DFPRS_Change_Cal_Table.ALL_plus
button at (980,231)-(1129,281): text "Decrease ALL"; taps DFPRS_Change_Cal_Table.ALL_minus
button at (1178,307)-(1320,387): text "Read Cal table"; taps DFPRS_Change_Cal_Table.Read_cal
button at (980,308)-(1138,376): text "Write Cal table"; taps DFPRS_Change_Cal_Table.Write_cal
button at (1175,155)-(1320,216): text "Set ALL"; taps DFPRS_Change_Cal_Table.Set_ALL
button at (1176,228)-(1321,281): text "HALF set  ALL"; taps DFPRS_Change_Cal_Table.HALF_set_ALL
button at (810,60)-(861,91): text "-"; taps DFPRS_Change_Cal_Table.RPM_Flag_minus_1
button at (740,100)-(791,131): text "+"; taps DFPRS_Change_Cal_Table.RPM_Flag_plus_2
button at (810,100)-(861,131): text "-"; taps DFPRS_Change_Cal_Table.RPM_Flag_minus_2
button at (880,100)-(931,131): text "CP 2"; taps DFPRS_Change_Cal_Table.RPM_Flag_CP_2
button at (740,140)-(791,171): text "+"; taps DFPRS_Change_Cal_Table.RPM_Flag_plus_3
button at (810,140)-(861,171): text "-"; taps DFPRS_Change_Cal_Table.RPM_Flag_minus_3
button at (880,140)-(931,171): text "CP 3"; taps DFPRS_Change_Cal_Table.RPM_Flag_CP_3
button at (740,180)-(791,211): text "+"; taps DFPRS_Change_Cal_Table.RPM_Flag_plus_4
button at (810,180)-(861,211): text "-"; taps DFPRS_Change_Cal_Table.RPM_Flag_minus_4
button at (880,180)-(931,211): text "CP 4"; taps DFPRS_Change_Cal_Table.RPM_Flag_CP_4
button at (740,220)-(791,251): text "+"; taps DFPRS_Change_Cal_Table.RPM_Flag_plus_5
button at (810,220)-(861,251): text "-"; taps DFPRS_Change_Cal_Table.RPM_Flag_minus_5
button at (880,220)-(931,251): text "CP 5"; taps DFPRS_Change_Cal_Table.RPM_Flag_CP_5
button at (740,255)-(791,286): text "+"; taps DFPRS_Change_Cal_Table.RPM_Flag_plus_6
button at (810,255)-(861,286): text "-"; taps DFPRS_Change_Cal_Table.RPM_Flag_minus_6
button at (880,255)-(931,286): text "CP 6"; taps DFPRS_Change_Cal_Table.RPM_Flag_CP_6
button at (740,295)-(791,326): text "+"; taps DFPRS_Change_Cal_Table.RPM_Flag_plus_7
button at (810,295)-(861,326): text "-"; taps DFPRS_Change_Cal_Table.RPM_Flag_minus_7
button at (880,295)-(931,326): text "CP 7"; taps DFPRS_Change_Cal_Table.RPM_Flag_CP_7
button at (740,330)-(791,361): text "+"; taps DFPRS_Change_Cal_Table.RPM_Flag_plus_8
button at (810,330)-(861,361): text "-"; taps DFPRS_Change_Cal_Table.RPM_Flag_minus_8
button at (880,330)-(931,361): text "CP 8"; taps DFPRS_Change_Cal_Table.RPM_Flag_CP_8
button at (90,675)-(121,696): text "+"; taps DFPRS_Change_Cal_Table.Turbo_Flag_plus_1
button at (90,705)-(121,726): text "-"; taps DFPRS_Change_Cal_Table.Turbo_Flag_minus_1
button at (130,675)-(161,696): text "+"; taps DFPRS_Change_Cal_Table.Turbo_Flag_plus_2
button at (130,705)-(161,726): text "-"; taps DFPRS_Change_Cal_Table.Turbo_Flag_minus_2
button at (128,736)-(159,757): text "CP2"; taps DFPRS_Change_Cal_Table.Turbo_Flag_CP_2
button at (170,675)-(201,696): text "+"; taps DFPRS_Change_Cal_Table.Turbo_Flag_plus_3
button at (170,705)-(201,726): text "-"; taps DFPRS_Change_Cal_Table.Turbo_Flag_minus_3
button at (168,736)-(199,757): text "CP3"; taps DFPRS_Change_Cal_Table.Turbo_Flag_CP_3
button at (210,675)-(241,696): text "+"; taps DFPRS_Change_Cal_Table.Turbo_Flag_plus_4
button at (210,705)-(241,726): text "-"; taps DFPRS_Change_Cal_Table.Turbo_Flag_minus_4
button at (208,736)-(239,757): text "CP4"; taps DFPRS_Change_Cal_Table.Turbo_Flag_CP_4
button at (250,675)-(281,696): text "+"; taps DFPRS_Change_Cal_Table.Turbo_Flag_plus_5
button at (250,705)-(281,726): text "-"; taps DFPRS_Change_Cal_Table.Turbo_Flag_minus_5
button at (248,736)-(279,757): text "CP5"; taps DFPRS_Change_Cal_Table.Turbo_Flag_CP_5
button at (295,675)-(326,696): text "+"; taps DFPRS_Change_Cal_Table.Turbo_Flag_plus_6
button at (295,705)-(326,726): text "-"; taps DFPRS_Change_Cal_Table.Turbo_Flag_minus_6
button at (293,736)-(324,757): text "CP6"; taps DFPRS_Change_Cal_Table.Turbo_Flag_CP_6
button at (335,675)-(366,696): text "+"; taps DFPRS_Change_Cal_Table.Turbo_Flag_plus_7
button at (335,705)-(366,726): text "-"; taps DFPRS_Change_Cal_Table.Turbo_Flag_minus_7
button at (333,736)-(364,757): text "CP7"; taps DFPRS_Change_Cal_Table.Turbo_Flag_CP_7
button at (375,675)-(406,696): text "+"; taps DFPRS_Change_Cal_Table.Turbo_Flag_plus_8
button at (375,705)-(406,726): text "-"; taps DFPRS_Change_Cal_Table.Turbo_Flag_minus_8
button at (373,736)-(404,757): text "CP8"; taps DFPRS_Change_Cal_Table.Turbo_Flag_CP_8
rounded rectangle at (1010,90)-(1264,141): text "Change value          %s"; shows DFPRS_Change_Cal_Table.Change_volume; editable 1..
rounded rectangle at (1175,400)-(1323,486): text "PPS / %s"; shows .PPS1
rounded rectangle at (1180,495)-(1325,581): text "HOLD / %s"; shows .Inj_PWM_time/4
rounded rectangle at (930,10)-(1296,71): text "GAS calibration table."
button at (990,590)-(1151,629): text "Read to buffer"; taps DFPRS_Change_Cal_Table.red_cal2
button at (990,640)-(1156,681): text "Write from buffer"; taps DFPRS_Change_Cal_Table.Write_cal2
rounded rectangle at (990,400)-(1138,486): text "RPM / %s"; shows .RPM
rounded rectangle at (995,495)-(1143,576): text "Turbo / %s"; shows .Turbo_pressure
rectangle at (0,0)-(0,0): text "%s"; shows p.PPS_table[1]; editable
rectangle at (0,0)-(0,0): text "%s"; shows p.PPS_table[2]; editable
rectangle at (0,0)-(0,0): text "%s"; shows p.PPS_table[3]; editable
rectangle at (0,0)-(0,0): text "%s"; shows p.PPS_table[4]; editable
rectangle at (0,0)-(0,0): text "%s"; shows p.PPS_table[5]; editable
rectangle at (0,0)-(0,0): text "%s"; shows p.PPS_table[6]; editable
rectangle at (0,0)-(0,0): text "%s"; shows p.PPS_table[7]; editable
rectangle at (0,0)-(0,0): text "%s"; shows p.PPS_table[8]; editable
rectangle at (0,0)-(0,0): text "%s"; shows p.PPS_table[9]; editable
rectangle at (0,0)-(0,0): text "%s"; shows p.PPS_table[10]; editable
rectangle at (0,0)-(0,0): text "%s"; shows p.PPS_table[11]; editable
rectangle at (0,0)-(0,0): text "%s"; shows p.PPS_table[12]; editable
rectangle at (0,0)-(0,0): text "%s"; shows p.PPS_table[13]; editable
rectangle at (0,0)-(0,0): text "%s"; shows p.PPS_table[14]; editable
rectangle at (0,0)-(0,0): text "%s"; shows p.PPS_table[15]; editable
rectangle at (0,0)-(0,0): text "%s"; shows p.PPS_table[16]; editable
rounded rectangle at (745,705)-(791,756): text "PPS"
button at (810,365)-(861,396): text "-"; taps DFPRS_Change_Cal_Table.RPM_Flag_minus_9
button at (740,405)-(791,436): text "+"; taps DFPRS_Change_Cal_Table.RPM_Flag_plus_10
button at (810,405)-(861,436): text "-"; taps DFPRS_Change_Cal_Table.RPM_Flag_minus_10
button at (880,405)-(931,436): text "CP 10"; taps DFPRS_Change_Cal_Table.RPM_Flag_CP_10
button at (740,445)-(791,476): text "+"; taps DFPRS_Change_Cal_Table.RPM_Flag_plus_11
button at (810,445)-(861,476): text "-"; taps DFPRS_Change_Cal_Table.RPM_Flag_minus_11
button at (880,445)-(931,476): text "CP 11"; taps DFPRS_Change_Cal_Table.RPM_Flag_CP_11
button at (740,485)-(791,516): text "+"; taps DFPRS_Change_Cal_Table.RPM_Flag_plus_12
button at (810,485)-(861,516): text "-"; taps DFPRS_Change_Cal_Table.RPM_Flag_minus_12
button at (880,485)-(931,516): text "CP 12"; taps DFPRS_Change_Cal_Table.RPM_Flag_CP_12
button at (740,525)-(791,556): text "+"; taps DFPRS_Change_Cal_Table.RPM_Flag_plus_13
button at (810,525)-(861,556): text "-"; taps DFPRS_Change_Cal_Table.RPM_Flag_minus_13
button at (880,525)-(931,556): text "CP 13"; taps DFPRS_Change_Cal_Table.RPM_Flag_CP_13
button at (740,560)-(791,591): text "+"; taps DFPRS_Change_Cal_Table.RPM_Flag_plus_14
button at (810,560)-(861,591): text "-"; taps DFPRS_Change_Cal_Table.RPM_Flag_minus_14
button at (880,560)-(931,591): text "CP 14"; taps DFPRS_Change_Cal_Table.RPM_Flag_CP_14
button at (740,600)-(791,631): text "+"; taps DFPRS_Change_Cal_Table.RPM_Flag_plus_15
button at (810,600)-(861,631): text "-"; taps DFPRS_Change_Cal_Table.RPM_Flag_minus_15
button at (880,600)-(931,631): text "CP 15"; taps DFPRS_Change_Cal_Table.RPM_Flag_CP_15
button at (740,635)-(791,666): text "+"; taps DFPRS_Change_Cal_Table.RPM_Flag_plus_16
button at (810,635)-(861,666): text "-"; taps DFPRS_Change_Cal_Table.RPM_Flag_minus_16
button at (880,635)-(931,666): text "CP 16"; taps DFPRS_Change_Cal_Table.RPM_Flag_CP_16
button at (880,365)-(931,396): text "CP 9"; taps DFPRS_Change_Cal_Table.RPM_Flag_CP_9
button at (415,675)-(446,696): text "+"; taps DFPRS_Change_Cal_Table.Turbo_Flag_plus_9
button at (415,705)-(446,726): text "-"; taps DFPRS_Change_Cal_Table.Turbo_Flag_minus_9
button at (455,675)-(486,696): text "+"; taps DFPRS_Change_Cal_Table.Turbo_Flag_plus_10
button at (455,705)-(486,726): text "-"; taps DFPRS_Change_Cal_Table.Turbo_Flag_minus_10
button at (453,736)-(491,757): text "CP10"; taps DFPRS_Change_Cal_Table.Turbo_Flag_CP_10
button at (495,675)-(526,696): text "+"; taps DFPRS_Change_Cal_Table.Turbo_Flag_plus_11
button at (495,705)-(526,726): text "-"; taps DFPRS_Change_Cal_Table.Turbo_Flag_minus_11
button at (493,736)-(526,757): text "CP11"; taps DFPRS_Change_Cal_Table.Turbo_Flag_CP_11
button at (535,675)-(566,696): text "+"; taps DFPRS_Change_Cal_Table.Turbo_Flag_plus_12
button at (535,705)-(566,726): text "-"; taps DFPRS_Change_Cal_Table.Turbo_Flag_minus_12
button at (533,736)-(571,757): text "CP12"; taps DFPRS_Change_Cal_Table.Turbo_Flag_CP_12
button at (575,675)-(606,696): text "+"; taps DFPRS_Change_Cal_Table.Turbo_Flag_plus_13
button at (575,705)-(606,726): text "-"; taps DFPRS_Change_Cal_Table.Turbo_Flag_minus_13
button at (573,736)-(611,757): text "CP13"; taps DFPRS_Change_Cal_Table.Turbo_Flag_CP_13
button at (620,675)-(651,696): text "+"; taps DFPRS_Change_Cal_Table.Turbo_Flag_plus_14
button at (620,705)-(651,726): text "-"; taps DFPRS_Change_Cal_Table.Turbo_Flag_minus_14
button at (618,736)-(651,757): text "CP14"; taps DFPRS_Change_Cal_Table.Turbo_Flag_CP_14
button at (660,675)-(691,696): text "+"; taps DFPRS_Change_Cal_Table.Turbo_Flag_plus_15
button at (660,705)-(691,726): text "-"; taps DFPRS_Change_Cal_Table.Turbo_Flag_minus_15
button at (658,736)-(691,757): text "CP15"; taps DFPRS_Change_Cal_Table.Turbo_Flag_CP_15
button at (700,675)-(731,696): text "+"; taps DFPRS_Change_Cal_Table.Turbo_Flag_plus_16
button at (700,705)-(731,726): text "-"; taps DFPRS_Change_Cal_Table.Turbo_Flag_minus_16
button at (698,736)-(731,757): text "CP16"; taps DFPRS_Change_Cal_Table.Turbo_Flag_CP_16
button at (415,735)-(446,756): text "CP9"; taps DFPRS_Change_Cal_Table.Turbo_Flag_CP_9
*)

(* Visualisation MAIN_PRIBOR
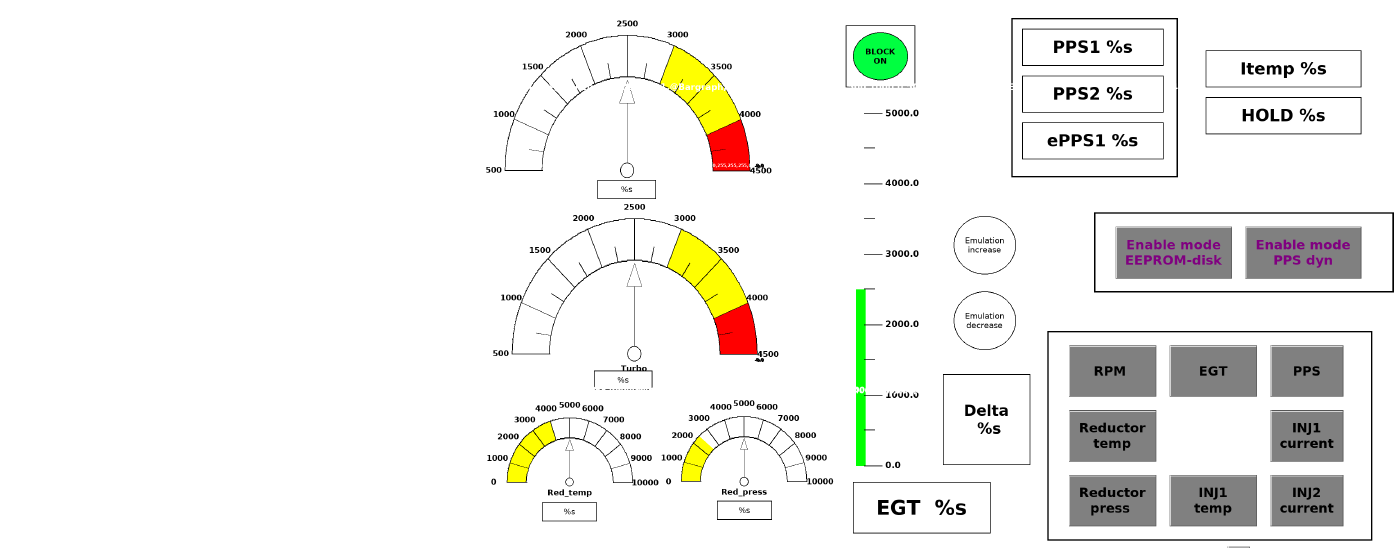
group at (15,5)-(416,256)
  rectangle at (0,0)-(1,1): text "{ExtendedElement},Visu\ElementDLL.ete,0,@Zeigerinstrument,401,180,0,0,255,255,255,0,RPM,RPM,%.0f,0,1,1,250,500,500,4500,0,0,0,0,0,0,0,-13,16,700,Arial,1,2,4000,4500,255,0,0,3000,4000,255,255,0,"
  rectangle at (5,192)-(26,208): text "500"
  rectangle at (16,122)-(44,138): text "1000"
  rectangle at (56,62)-(84,78): text "1500"
  rectangle at (116,22)-(144,38): text "2000"
  rectangle at (187,8)-(215,24): text "2500"
  rectangle at (257,22)-(285,38): text "3000"
  rectangle at (317,62)-(345,78): text "3500"
  rectangle at (357,122)-(385,138): text "4000"
  rectangle at (372,193)-(400,209): text "4500"
  rectangle at (186,211)-(215,227): text "RPM"
  polygon at (190,87)-(211,201): angle ((RPM * 1.0)-2500) * 0.045
group at (400,220)-(401,221)
  rectangle at (0,0)-(1,1): text "{ExtendedElement},Visu\ElementDLL.ete,0,@Zeigerinstrument,200,180,0,0,255,255,255,0,,,%.1f,0,1,1,1,2,-4,4,0,0,0,0,0,0,0,-13,16,700,Arial,1,2,4000,5500,255,255,128,5500,6000,255,0,0,"
  rectangle at (1,92)-(23,108): text "-4.0"
  rectangle at (27,30)-(49,46): text "-2.0"
  rectangle at (91,4)-(109,20): text "0.0"
  rectangle at (153,30)-(171,46): text "2.0"
  rectangle at (179,92)-(197,108): text "4.0"
group at (400,490)-(401,491)
  rectangle at (0,0)-(1,1): text "{ExtendedElement},Visu\ElementDLL.ete,0,@Zeigerinstrument,200,180,0,0,255,255,255,0,,,%.1f,0,1,1,1,2,-4,4,0,0,0,0,0,0,0,-13,16,700,Arial,1,2,4000,5500,255,255,128,5500,6000,255,0,0,"
  rectangle at (1,92)-(23,108): text "-4.0"
  rectangle at (27,30)-(49,46): text "-2.0"
  rectangle at (91,4)-(109,20): text "0.0"
  rectangle at (153,30)-(171,46): text "2.0"
  rectangle at (179,92)-(197,108): text "4.0"
group at (25,260)-(426,511)
  rectangle at (0,0)-(1,1): text "{ExtendedElement},Visu\ElementDLL.ete,0,@Zeigerinstrument,401,180,0,0,255,255,255,0,Turbo_pressure,Turbo,%.0f,0,1,1,250,500,500,4500,0,0,0,0,0,0,0,-13,16,700,Arial,1,2,3000,4000,255,255,0,4000,4500,255,0,0,"
  rectangle at (5,192)-(26,208): text "500"
  rectangle at (16,122)-(44,138): text "1000"
  rectangle at (56,62)-(84,78): text "1500"
  rectangle at (116,22)-(144,38): text "2000"
  rectangle at (187,8)-(215,24): text "2500"
  rectangle at (257,22)-(285,38): text "3000"
  rectangle at (317,62)-(345,78): text "3500"
  rectangle at (357,122)-(385,138): text "4000"
  rectangle at (372,193)-(400,209): text "4500"
  rectangle at (182,211)-(219,227): text "Turbo"
  polygon at (190,87)-(211,201): angle ((Turbo_pressure * 1.0)-2500) * 0.045
rounded rectangle at (170,505)-(251,531): text "%s"; shows .Turbo_pressure
rounded rectangle at (175,240)-(256,266): text "%s"; shows .RPM
group at (515,110)-(626,648)
  rectangle at (0,0)-(1,1): text "{ExtendedElement},Visu\ElementDLL.ete,1,@Bargraph,101,511,0,1,0,EGT,,%.1f,500,1000,0,5000,0,0,0,0,0,0,0,-13,16,700,Arial,0,255,0,255,0,0,1,4500,0,0,0,"
  rectangle at (16,255)-(27,476): alarm colour if (EGT) > 4500; top ((EGT * 1.0) - 2500)  * -0.0884
  rectangle at (49,465)-(94,486): text "0.0"
  rectangle at (49,377)-(94,398): text "1000.0"
  rectangle at (49,288)-(94,309): text "2000.0"
  rectangle at (49,200)-(94,221): text "3000.0"
  rectangle at (49,111)-(94,132): text "4000.0"
  rectangle at (49,23)-(94,44): text "5000.0"
group at (11,532)-(259,683)
  rectangle at (0,0)-(1,1): text "{ExtendedElement},Visu\ElementDLL.ete,0,@Zeigerinstrument,249,180,0,0,255,255,255,0,Reductor_temp,Red_temp,%.0f,0,1,1,1000,1000,0,10000,0,0,0,0,0,0,0,-13,16,700,Arial,1,1,0,4000,255,255,0,"
  rectangle at (16,116)-(23,133): text "0"
  rectangle at (11,84)-(39,100): text "1000"
  rectangle at (26,55)-(54,71): text "2000"
  rectangle at (49,32)-(77,48): text "3000"
  rectangle at (78,17)-(106,33): text "4000"
  rectangle at (111,12)-(139,28): text "5000"
  rectangle at (143,17)-(171,33): text "6000"
  rectangle at (172,32)-(200,48): text "7000"
  rectangle at (195,55)-(223,71): text "8000"
  rectangle at (210,84)-(238,100): text "9000"
  rectangle at (212,117)-(247,133): text "10000"
  rectangle at (93,131)-(157,147): text "Red_temp"
  polygon at (119,67)-(130,125): angle ((Reductor_temp * 1.0)-5000) * 0.018
rounded rectangle at (98,688)-(174,714): text "%s"; shows .Reductor_temp
rounded rectangle at (530,660)-(721,731): text "EGT  %s"; shows .EGT
ellipse at (530,35)-(606,101): text "BLOCK / ON"; alarm colour if .Flag_ECU_ON=FALSE
rounded rectangle at (1020,125)-(1236,176): text "HOLD %s"; shows .Inj_PWM_time/4
group at (254,531)-(502,682)
  rectangle at (0,0)-(1,1): text "{ExtendedElement},Visu\ElementDLL.ete,0,@Zeigerinstrument,248,180,0,0,255,255,255,0,Reductor_press,Red_press,%.0f,0,1,1,1000,1000,0,10000,0,0,0,0,0,0,0,-13,16,700,Arial,1,1,0,2500,255,255,0,"
  rectangle at (16,116)-(23,132): text "0"
  rectangle at (10,84)-(38,100): text "1000"
  rectangle at (25,54)-(53,70): text "2000"
  rectangle at (48,31)-(76,47): text "3000"
  rectangle at (78,16)-(106,32): text "4000"
  rectangle at (110,11)-(138,27): text "5000"
  rectangle at (142,16)-(170,32): text "6000"
  rectangle at (172,31)-(200,47): text "7000"
  rectangle at (195,54)-(223,70): text "8000"
  rectangle at (210,84)-(238,100): text "9000"
  rectangle at (212,116)-(247,132): text "10000"
  rectangle at (92,130)-(157,146): text "Red_press"
  polygon at (119,66)-(129,124): angle ((Reductor_press * 1.0)-5000) * 0.018
rounded rectangle at (341,686)-(417,712): text "%s"; shows .Reductor_press
rounded rectangle at (1020,60)-(1236,111): text "Itemp %s"; shows .Injector_temp
rounded rectangle at (765,30)-(961,81): text "PPS1 %s"; shows .PPS1
rounded rectangle at (765,95)-(961,146): text "PPS2 %s"; shows .PPS2
rounded rectangle at (765,160)-(961,211): text "ePPS1 %s"; shows .PPS1_emul
button at (1075,305)-(1236,377): text "Enable mode / PPS dyn"; toggles .Flag_PPS_dyn_enable
button at (830,470)-(951,541): text "RPM"; toggles .Err_RPM
button at (970,470)-(1091,541): text "EGT"; toggles .Err_EGT
button at (830,560)-(951,631): text "Reductor / temp"; toggles .Err_Reductor_temp
button at (830,650)-(951,721): text "Reductor / press"; shows .Reductor_press; toggles .Err_Reductor_press
button at (1110,560)-(1211,631): text "INJ1 / current"; toggles .Err_Inj1
button at (1110,650)-(1211,721): text "INJ2 / current"; toggles .Err_Inj2
button at (970,650)-(1091,721): text "INJ1 / temp"; toggles .Err_Inj_temp
button at (1110,470)-(1211,541): text "PPS"; toggles .Err_PPS
ellipse at (670,290)-(756,371): text "Emulation / increase"; alarm colour if Act_control.Flag_PPS_plus=FALSE
button at (895,305)-(1056,377): text "Enable mode / EEPROM-disk"; toggles .Flag_CAN
ellipse at (670,395)-(756,476): text "Emulation / decrease"; alarm colour if Act_control.Flag_PPS_minus=FALSE
rounded rectangle at (655,510)-(776,636): text "Delta / %s"; shows Act_control.delta
116 more shapes without text or variables
*)
